	{attribute 'TcIecLibraryType'}
	{attribute 'external_name' := 'F_VN_CreateBandpassButterworthFilter_GUID_D3DC1E0E_00A6_3CD1_3172_0A7CC9A7F473'}
	(* Creates a bandpass Butterworth filter, which can be applied to a frequency domain image by element-wise multiplication. *)
	FUNCTION F_VN_CreateBandpassButterworthFilter : HRESULT
	VAR_INPUT
		ipFilter	:	REFERENCE TO ITcVnImage;	(* Returns the created filter (1 channel of type REAL or LREAL, depending on bDoublePrecision. Non-zero interface pointers are reused.). *)
		nWidth	:	UDINT;	(* Filter width (even, >= 2, must match the width of the image it is applied to) *)
		nHeight	:	UDINT;	(* Filter height (even, >= 2, must match the height of the image it is applied to) *)
		bDoublePrecision	:	BOOL;	(* If true, the filter is generated with double precision (LREAL) instead of single precision (REAL). *)
		bOriginAtCenter	:	BOOL;	(* If true, the filter origin is shifted to the image center. *)
		fCutoffDistance	:	LREAL;	(* The cutoff distance of the Butterworth filter (> 0). *)
		fBandWidth	:	LREAL;	(* The band width of the Butterworth filter (> 0). *)
		nOrder	:	UDINT;	(* The order of the Butterworth filter (> 0). *)
		fScale	:	LREAL;	(* The scale factor of the Butterworth filter denominator term (> 0, e.g. 0.414 or 1.0). *)
		hrPrev	:	HRESULT;	(* HRESULT indicating the result of previous operations (If SUCCEEDED(hrPrev) equals false, no operation is executed.) *)
	END_VAR

END_FUNCTION

// Functions/Fourier Analysis/F_VN_CreateBandpassGaussianFilter

	{attribute 'TcIecLibraryType'}
	{attribute 'external_name' := 'F_VN_CreateBandpassGaussianFilter_GUID_DC938AC3_3255_3FAF_03A0_1C1517F5338C'}
	(* Creates a bandpass Gaussian filter, which can be applied to a frequency domain image by element-wise multiplication. *)
	FUNCTION F_VN_CreateBandpassGaussianFilter : HRESULT
	VAR_INPUT
		ipFilter	:	REFERENCE TO ITcVnImage;	(* Returns the created filter (1 channel of type REAL or LREAL, depending on bDoublePrecision. Non-zero interface pointers are reused.). *)
		nWidth	:	UDINT;	(* Filter width (even, >= 2, must match the width of the image it is applied to) *)
		nHeight	:	UDINT;	(* Filter height (even, >= 2, must match the height of the image it is applied to) *)
		bDoublePrecision	:	BOOL;	(* If true, the filter is generated with double precision (LREAL) instead of single precision (REAL). *)
		bOriginAtCenter	:	BOOL;	(* If true, the filter origin is shifted to the image center. *)
		fCutoffDistance	:	LREAL;	(* The cutoff distance of the Gaussian filter (> 0). *)
		fBandWidth	:	LREAL;	(* The band width of the Gaussian filter (> 0). *)
		hrPrev	:	HRESULT;	(* HRESULT indicating the result of previous operations (If SUCCEEDED(hrPrev) equals false, no operation is executed.) *)
	END_VAR

END_FUNCTION

// Functions/Fourier Analysis/F_VN_CreateBandrejectButterworthFilter

	{attribute 'TcIecLibraryType'}
	{attribute 'external_name' := 'F_VN_CreateBandrejectButterworthFilter_GUID_34508946_AADD_3D36_1DBA_977273E9C532'}
	(* Creates a bandreject Butterworth filter, which can be applied to a frequency domain image by element-wise multiplication. *)
	FUNCTION F_VN_CreateBandrejectButterworthFilter : HRESULT
	VAR_INPUT
		ipFilter	:	REFERENCE TO ITcVnImage;	(* Returns the created filter (1 channel of type REAL or LREAL, depending on bDoublePrecision. Non-zero interface pointers are reused.). *)
		nWidth	:	UDINT;	(* Filter width (even, >= 2, must match the width of the image it is applied to) *)
		nHeight	:	UDINT;	(* Filter height (even, >= 2, must match the height of the image it is applied to) *)
		bDoublePrecision	:	BOOL;	(* If true, the filter is generated with double precision (LREAL) instead of single precision (REAL). *)
		bOriginAtCenter	:	BOOL;	(* If true, the filter origin is shifted to the image center. *)
		fCutoffDistance	:	LREAL;	(* The cutoff distance of the Butterworth filter (> 0). *)
		fBandWidth	:	LREAL;	(* The band width of the Butterworth filter (> 0). *)
		nOrder	:	UDINT;	(* The order of the Butterworth filter (> 0). *)
		fScale	:	LREAL;	(* The scale factor of the Butterworth filter denominator term (> 0, e.g. 0.414 or 1.0). *)
		hrPrev	:	HRESULT;	(* HRESULT indicating the result of previous operations (If SUCCEEDED(hrPrev) equals false, no operation is executed.) *)
	END_VAR

END_FUNCTION

// Functions/Fourier Analysis/F_VN_CreateBandrejectGaussianFilter

	{attribute 'TcIecLibraryType'}
	{attribute 'external_name' := 'F_VN_CreateBandrejectGaussianFilter_GUID_5AAE8B01_5460_3F06_0DD8_D2F7DBC7A3F1'}
	(* Creates a bandreject Gaussian filter, which can be applied to a frequency domain image by element-wise multiplication. *)
	FUNCTION F_VN_CreateBandrejectGaussianFilter : HRESULT
	VAR_INPUT
		ipFilter	:	REFERENCE TO ITcVnImage;	(* Returns the created filter (1 channel of type REAL or LREAL, depending on bDoublePrecision. Non-zero interface pointers are reused.). *)
		nWidth	:	UDINT;	(* Filter width (even, >= 2, must match the width of the image it is applied to) *)
		nHeight	:	UDINT;	(* Filter height (even, >= 2, must match the height of the image it is applied to) *)
		bDoublePrecision	:	BOOL;	(* If true, the filter is generated with double precision (LREAL) instead of single precision (REAL). *)
		bOriginAtCenter	:	BOOL;	(* If true, the filter origin is shifted to the image center. *)
		fCutoffDistance	:	LREAL;	(* The cutoff distance of the Gaussian filter (> 0). *)
		fBandWidth	:	LREAL;	(* The band width of the Gaussian filter (> 0). *)
		hrPrev	:	HRESULT;	(* HRESULT indicating the result of previous operations (If SUCCEEDED(hrPrev) equals false, no operation is executed.) *)
	END_VAR

END_FUNCTION

// Functions/Fourier Analysis/F_VN_CreateHighpassButterworthFilter

	{attribute 'TcIecLibraryType'}
	{attribute 'external_name' := 'F_VN_CreateHighpassButterworthFilter_GUID_519CDF3B_54D9_3152_1A44_7AA98764909A'}
	(* Creates a highpass Butterworth filter, which can be applied to a frequency domain image by element-wise multiplication. *)
	FUNCTION F_VN_CreateHighpassButterworthFilter : HRESULT
	VAR_INPUT
		ipFilter	:	REFERENCE TO ITcVnImage;	(* Returns the created filter (1 channel of type REAL or LREAL, depending on bDoublePrecision. Non-zero interface pointers are reused.). *)
		nWidth	:	UDINT;	(* Filter width (even, >= 2, must match the width of the image it is applied to) *)
		nHeight	:	UDINT;	(* Filter height (even, >= 2, must match the height of the image it is applied to) *)
		bDoublePrecision	:	BOOL;	(* If true, the filter is generated with double precision (LREAL) instead of single precision (REAL). *)
		bOriginAtCenter	:	BOOL;	(* If true, the filter origin is shifted to the image center. *)
		fCutoffDistance	:	LREAL;	(* The cutoff distance of the Butterworth filter (> 0). *)
		nOrder	:	UDINT;	(* The order of the Butterworth filter (> 0). *)
		fScale	:	LREAL;	(* The scale factor of the Butterworth filter denominator term (> 0, e.g. 0.414 or 1.0). *)
		hrPrev	:	HRESULT;	(* HRESULT indicating the result of previous operations (If SUCCEEDED(hrPrev) equals false, no operation is executed.) *)
	END_VAR

END_FUNCTION

// Functions/Fourier Analysis/F_VN_CreateHighpassGaussianFilter

	{attribute 'TcIecLibraryType'}
	{attribute 'external_name' := 'F_VN_CreateHighpassGaussianFilter_GUID_E618411A_DEFA_3D5F_3B14_5E90FD46016B'}
	(* Creates a highpass Gaussian filter, which can be applied to a frequency domain image by element-wise multiplication. *)
	FUNCTION F_VN_CreateHighpassGaussianFilter : HRESULT
	VAR_INPUT
		ipFilter	:	REFERENCE TO ITcVnImage;	(* Returns the created filter (1 channel of type REAL or LREAL, depending on bDoublePrecision. Non-zero interface pointers are reused.). *)
		nWidth	:	UDINT;	(* Filter width (even, >= 2, must match the width of the image it is applied to) *)
		nHeight	:	UDINT;	(* Filter height (even, >= 2, must match the height of the image it is applied to) *)
		bDoublePrecision	:	BOOL;	(* If true, the filter is generated with double precision (LREAL) instead of single precision (REAL). *)
		bOriginAtCenter	:	BOOL;	(* If true, the filter origin is shifted to the image center. *)
		fCutoffDistance	:	LREAL;	(* The cutoff distance of the Gaussian filter (> 0). *)
		hrPrev	:	HRESULT;	(* HRESULT indicating the result of previous operations (If SUCCEEDED(hrPrev) equals false, no operation is executed.) *)
	END_VAR

END_FUNCTION

// Functions/Fourier Analysis/F_VN_CreateLowpassButterworthFilter

	{attribute 'TcIecLibraryType'}
	{attribute 'external_name' := 'F_VN_CreateLowpassButterworthFilter_GUID_409D1272_0EF9_3A29_163E_A5ADC220BBB4'}
	(* Creates a lowpass Butterworth filter, which can be applied to a frequency domain image by element-wise multiplication. *)
	FUNCTION F_VN_CreateLowpassButterworthFilter : HRESULT
	VAR_INPUT
		ipFilter	:	REFERENCE TO ITcVnImage;	(* Returns the created filter (1 channel of type REAL or LREAL, depending on bDoublePrecision. Non-zero interface pointers are reused.). *)
		nWidth	:	UDINT;	(* Filter width (even, >= 2, must match the width of the image it is applied to) *)
		nHeight	:	UDINT;	(* Filter height (even, >= 2, must match the height of the image it is applied to) *)
		bDoublePrecision	:	BOOL;	(* If true, the filter is generated with double precision (LREAL) instead of single precision (REAL). *)
		bOriginAtCenter	:	BOOL;	(* If true, the filter origin is shifted to the image center. *)
		fCutoffDistance	:	LREAL;	(* The cutoff distance of the Butterworth filter (> 0). *)
		nOrder	:	UDINT;	(* The order of the Butterworth filter (> 0). *)
		fScale	:	LREAL;	(* The scale factor of the Butterworth filter denominator term (> 0, e.g. 0.414 or 1.0). *)
		hrPrev	:	HRESULT;	(* HRESULT indicating the result of previous operations (If SUCCEEDED(hrPrev) equals false, no operation is executed.) *)
	END_VAR

END_FUNCTION

// Functions/Fourier Analysis/F_VN_CreateLowpassGaussianFilter

	{attribute 'TcIecLibraryType'}
	{attribute 'external_name' := 'F_VN_CreateLowpassGaussianFilter_GUID_8B9BD84E_306C_3412_3556_4171BB31A9AA'}
	(* Creates a lowpass Gaussian filter, which can be applied to a frequency domain image by element-wise multiplication. *)
	FUNCTION F_VN_CreateLowpassGaussianFilter : HRESULT
	VAR_INPUT
		ipFilter	:	REFERENCE TO ITcVnImage;	(* Returns the created filter (1 channel of type REAL or LREAL, depending on bDoublePrecision. Non-zero interface pointers are reused.). *)
		nWidth	:	UDINT;	(* Filter width (even, >= 2, must match the width of the image it is applied to) *)
		nHeight	:	UDINT;	(* Filter height (even, >= 2, must match the height of the image it is applied to) *)
		bDoublePrecision	:	BOOL;	(* If true, the filter is generated with double precision (LREAL) instead of single precision (REAL). *)
		bOriginAtCenter	:	BOOL;	(* If true, the filter origin is shifted to the image center. *)
		fCutoffDistance	:	LREAL;	(* The cutoff distance of the Gaussian filter (> 0). *)
		hrPrev	:	HRESULT;	(* HRESULT indicating the result of previous operations (If SUCCEEDED(hrPrev) equals false, no operation is executed.) *)
	END_VAR

END_FUNCTION

// Functions/Fourier Analysis/F_VN_Dft

	{attribute 'TcIecLibraryType'}
	{attribute 'external_name' := 'F_VN_Dft_GUID_EB7F674C_B2FA_362B_333C_E819879DB455'}
	(* Computes the DFT for a given image. *)
	FUNCTION F_VN_Dft : HRESULT
	VAR_INPUT
		ipSpatialImage	:	ITcVnImage;	(* Source image (elements of type REAL or LREAL, 1 (Re) or 2 (Re + Im) channels) *)
		ipFrequencyImage	:	REFERENCE TO ITcVnImage;	(* Destination image (same type as ipSpatialImage, but number of channels and size can vary depending on bPackedCCS and bAutoPadding. *)
		bPackedCCS	:	BOOL;	(* If true and ipSpatialImage has only 1 channel, the result image will have 1 channel with packed complex-conjugate-symmetrical format results. Otherwise, the result image will have 2 separate channels (Re + Im), containing the full spectrum. *)
		bAutoPadding	:	BOOL;	(* If true, the input image is automatically padded (with 0s) to optimal size if required, to speed up dft (Creates a temporary copy so that ipSpatialImage content stays unchanged, which also requires some additional computation power. Therefore, it is recommended to compare execution times with and without padding.) *)
		hrPrev	:	HRESULT;	(* HRESULT indicating the result of previous operations (If SUCCEEDED(hrPrev) equals false, no operation is executed.) *)
	END_VAR

END_FUNCTION

// Functions/Fourier Analysis/F_VN_InverseDft

	{attribute 'TcIecLibraryType'}
	{attribute 'external_name' := 'F_VN_InverseDft_GUID_263D4574_0F7D_3790_12C2_708D290903E7'}
	(* Compute the inverse DFT for a given frequency image. *)
	FUNCTION F_VN_InverseDft : HRESULT
	VAR_INPUT
		ipFrequencyImage	:	ITcVnImage;	(* Source frequency image (elements of type REAL or LREAL, 1 (packed CCS) or 2 (Re + Im) channels) *)
		ipSpatialImage	:	REFERENCE TO ITcVnImage;	(* Destination image (Same type as ipFrequencyImage, but number of channels can vary depending on bRealOutput. An appropriate image will be created if required.) *)
		bRealOutput	:	BOOL;	(* Only relevant if ipFrequencyImage has 2 channels. If true, the result image will have only 1 channel. Otherwise, the result image will have 2 separate channels (Re + Im). If ipFrequencyImage has only 1 channel, packed CCS format is assumed and the result image will always have only 1 channel. *)
		hrPrev	:	HRESULT;	(* HRESULT indicating the result of previous operations (If SUCCEEDED(hrPrev) equals false, no operation is executed.) *)
	END_VAR

END_FUNCTION

// Functions/Fourier Analysis/F_VN_OptimalDftSize

	{attribute 'TcIecLibraryType'}
	{attribute 'external_name' := 'F_VN_OptimalDftSize_GUID_08DF2A98_D3C0_3961_2808_BBB884F661F3'}
	(* Computes the optimal image size for applying a dft (can lead to better performance). *)
	FUNCTION F_VN_OptimalDftSize : HRESULT
	VAR_INPUT
		ipImage	:	ITcVnImage;	(* Source image for which to compute the optimal width and height *)
		nOptWidth	:	REFERENCE TO UDINT;	(* Returns the optimal width of the image *)
		nOptHeight	:	REFERENCE TO UDINT;	(* Returns the optimal height of the image *)
		hrPrev	:	HRESULT;	(* HRESULT indicating the result of previous operations (If SUCCEEDED(hrPrev) equals false, no operation is executed.) *)
	END_VAR

END_FUNCTION

// Functions/Fourier Analysis/F_VN_PadImageBorder

	{attribute 'TcIecLibraryType'}
	{attribute 'external_name' := 'F_VN_PadImageBorder_GUID_7562E341_2B8B_34BB_14E9_157BF85E1FEC'}
	(* Add padding (zeros) around the original image borders. *)
	FUNCTION F_VN_PadImageBorder : HRESULT
	VAR_INPUT
		ipSrcImage	:	ITcVnImage;	(* Source image *)
		ipPaddedImage	:	REFERENCE TO ITcVnImage;	(* Padded destination image (Same type as ipSrcImage, an appropriate destination image will be created if required.) *)
		nTopBorder	:	UDINT;	(* Padding height in pixels above top border *)
		nBottomBorder	:	UDINT;	(* Padding height in pixels below bottom border *)
		nLeftBorder	:	UDINT;	(* Padding width in pixels before left border *)
		nRightBorder	:	UDINT;	(* Padding width in pixels after right border *)
		hrPrev	:	HRESULT;	(* HRESULT indicating the result of previous operations (If SUCCEEDED(hrPrev) equals false, no operation is executed.) *)
	END_VAR

END_FUNCTION

// Functions/Fourier Analysis/F_VN_PadImageBorderExp

	{attribute 'TcIecLibraryType'}
	{attribute 'external_name' := 'F_VN_PadImageBorderExp_GUID_D24854F6_1D3E_319C_162B_E66C409C6D41'}
	(* Add padding around the original image borders. (expert function) *)
	FUNCTION F_VN_PadImageBorderExp : HRESULT
	VAR_INPUT
		ipSrcImage	:	ITcVnImage;	(* Source image *)
		ipPaddedImage	:	REFERENCE TO ITcVnImage;	(* Padded destination image (Same type as ipSrcImage, an appropriate destination image will be created if required.) *)
		nTopBorder	:	UDINT;	(* Padding height in pixels above top border *)
		nBottomBorder	:	UDINT;	(* Padding height in pixels below bottom border *)
		nLeftBorder	:	UDINT;	(* Padding width in pixels before left border *)
		nRightBorder	:	UDINT;	(* Padding width in pixels after right border *)
		ePaddingType	:	ETcVnBorderInterpolationMethod;	(* Specifies how the pixel values of the padding area are determined *)
		aPaddingValue	:	REFERENCE TO TcVnVector4_LREAL;	(* Specifies the padding value if CONSTANT is used *)
		hrPrev	:	HRESULT;	(* HRESULT indicating the result of previous operations (If SUCCEEDED(hrPrev) equals false, no operation is executed.) *)
	END_VAR

END_FUNCTION

// Functions/Drawing/F_VN_DrawCircle

	{attribute 'TcIecLibraryType'}
	{attribute 'external_name' := 'F_VN_DrawCircle_GUID_1503D671_B32A_39B0_1A7E_BB6D47FEB820'}
	(* Draws a circle. *)
	FUNCTION F_VN_DrawCircle : HRESULT
	VAR_INPUT
		nCenterX	:	UDINT;	(* x coordinate of the center *)
		nCenterY	:	UDINT;	(* y coordinate of the center *)
		nRadius	:	UDINT;	(* Radius *)
		ipDestImage	:	ITcVnImage;	(* Destination image *)
		aColor	:	REFERENCE TO TcVnVector4_LREAL;	(* Color *)
		nThickness	:	DINT;	(* Line thickness (if negative, the circle is filled) *)
		hrPrev	:	HRESULT;	(* HRESULT indicating the result of previous operations (If SUCCEEDED(hrPrev) equals false, no operation is executed.) *)
	END_VAR

END_FUNCTION

// Functions/Drawing/F_VN_DrawCircleExp

	{attribute 'TcIecLibraryType'}
	{attribute 'external_name' := 'F_VN_DrawCircleExp_GUID_1BBCEDF2_9DF7_3314_302A_7B7B49323D97'}
	(* Draws a circle. *)
	FUNCTION F_VN_DrawCircleExp : HRESULT
	VAR_INPUT
		nCenterX	:	UDINT;	(* x coordinate of the center *)
		nCenterY	:	UDINT;	(* y coordinate of the center *)
		nRadius	:	UDINT;	(* Radius *)
		ipDestImage	:	ITcVnImage;	(* Destination image *)
		aColor	:	REFERENCE TO TcVnVector4_LREAL;	(* Color *)
		nThickness	:	DINT;	(* Line thickness (if negative, the circle is filled) *)
		eLineType	:	ETcVnLineType;	(* Line type *)
		hrPrev	:	HRESULT;	(* HRESULT indicating the result of previous operations (If SUCCEEDED(hrPrev) equals false, no operation is executed.) *)
	END_VAR

END_FUNCTION

// Functions/Drawing/F_VN_DrawCircles

	{attribute 'TcIecLibraryType'}
	{attribute 'external_name' := 'F_VN_DrawCircles_GUID_E3A7DD5D_261F_3C34_1E11_9BA2656FD439'}
	(* Draws circles. *)
	FUNCTION F_VN_DrawCircles : HRESULT
	VAR_INPUT
		ipCircles	:	ITcVnContainer;	(* Container with circles (ContainerType_Vector_TcVnVector3_REAL; Each container element contains the x coordinate of the circle center [0], the y coordinate of the circle center [1], and the radius [2].) *)
		nCircleIndex	:	DINT;	(* Index of a specific circle to be drawn (if negative, all circles within the container are drawn) *)
		ipDestImage	:	ITcVnImage;	(* Destination image *)
		aColor	:	REFERENCE TO TcVnVector4_LREAL;	(* Color *)
		nThickness	:	DINT;	(* Line thickness (if negative, the circle is filled) *)
		hrPrev	:	HRESULT;	(* HRESULT indicating the result of previous operations (If SUCCEEDED(hrPrev) equals false, no operation is executed.) *)
	END_VAR

END_FUNCTION

// Functions/Drawing/F_VN_DrawCirclesExp

	{attribute 'TcIecLibraryType'}
	{attribute 'external_name' := 'F_VN_DrawCirclesExp_GUID_B0C9EA54_3854_3F37_1BB4_4F32EA6C7A2F'}
	(* Draws circles. (expert function) *)
	FUNCTION F_VN_DrawCirclesExp : HRESULT
	VAR_INPUT
		ipCircles	:	ITcVnContainer;	(* Container with circles (ContainerType_Vector_TcVnVector3_REAL; Each container element contains the x coordinate of the circle center [0], the y coordinate of the circle center [1], and the radius [2].) *)
		nCircleIndex	:	DINT;	(* Index of a specific circle to be drawn (if negative, all circles within the container are drawn) *)
		ipDestImage	:	ITcVnImage;	(* Destination image *)
		aColor	:	REFERENCE TO TcVnVector4_LREAL;	(* Color *)
		nThickness	:	DINT;	(* Line thickness (if negative, the circle is filled) *)
		eLineType	:	ETcVnLineType;	(* Line type *)
		hrPrev	:	HRESULT;	(* HRESULT indicating the result of previous operations (If SUCCEEDED(hrPrev) equals false, no operation is executed.) *)
	END_VAR

END_FUNCTION

// Functions/Drawing/F_VN_DrawCircularArc

	{attribute 'TcIecLibraryType'}
	{attribute 'external_name' := 'F_VN_DrawCircularArc_GUID_121719E0_05DB_3D67_0B75_713630B18D92'}
	(* Draws a circular arc. *)
	FUNCTION F_VN_DrawCircularArc : HRESULT
	VAR_INPUT
		stCircularArc	:	REFERENCE TO TcVnCircularArc;	(* Circular arc definition *)
		ipDestImage	:	ITcVnImage;	(* Destination image *)
		aColor	:	REFERENCE TO TcVnVector4_LREAL;	(* Color *)
		nThickness	:	DINT;	(* Line thickness (if negative, the arc is filled) *)
		hrPrev	:	HRESULT;	(* HRESULT indicating the result of previous operations (If SUCCEEDED(hrPrev) equals false, no operation is executed.) *)
	END_VAR

END_FUNCTION

// Functions/Drawing/F_VN_DrawCircularArcExp

	{attribute 'TcIecLibraryType'}
	{attribute 'external_name' := 'F_VN_DrawCircularArcExp_GUID_29FE52B3_2C94_302D_17C7_3DEA0BEF895C'}
	(* Draws a circular arc. (expert function) *)
	FUNCTION F_VN_DrawCircularArcExp : HRESULT
	VAR_INPUT
		stCircularArc	:	REFERENCE TO TcVnCircularArc;	(* Circular arc definition *)
		ipDestImage	:	ITcVnImage;	(* Destination image *)
		aColor	:	REFERENCE TO TcVnVector4_LREAL;	(* Color *)
		nThickness	:	DINT;	(* Line thickness (if negative, the arc is filled) *)
		eLineType	:	ETcVnLineType;	(* Line type *)
		hrPrev	:	HRESULT;	(* HRESULT indicating the result of previous operations (If SUCCEEDED(hrPrev) equals false, no operation is executed.) *)
	END_VAR

END_FUNCTION

// Functions/Drawing/F_VN_DrawContours

	{attribute 'TcIecLibraryType'}
	{attribute 'external_name' := 'F_VN_DrawContours_GUID_4DDB8EE0_9EFD_3D7D_0A1D_A16515665A8A'}
	(* Draws a single point set or multiple point sets that are interpreted as contours. *)
	FUNCTION F_VN_DrawContours : HRESULT
	VAR_INPUT
		ipContours	:	ITcVnContainer;	(* Single contour (ContainerType_Vector_TcVnPoint2_DINT) or multiple contours (ContainerType_Vector_Vector_TcVnPoint2_DINT) *)
		nContourIndex	:	DINT;	(* Index of a specific contour to be drawn (if negative, all contours within the container are drawn) *)
		ipDestImage	:	ITcVnImage;	(* Destination image *)
		aColor	:	REFERENCE TO TcVnVector4_LREAL;	(* Color *)
		nThickness	:	DINT;	(* Line thickness (if negative, the contours are filled) *)
		hrPrev	:	HRESULT;	(* HRESULT indicating the result of previous operations (If SUCCEEDED(hrPrev) equals false, no operation is executed.) *)
	END_VAR

END_FUNCTION

// Functions/Drawing/F_VN_DrawContoursExp

	{attribute 'TcIecLibraryType'}
	{attribute 'external_name' := 'F_VN_DrawContoursExp_GUID_3EB6DE25_2DBC_399F_1688_26782D4E7652'}
	(* Draws a single point set or multiple point sets that are interpreted as contours. (expert function) *)
	FUNCTION F_VN_DrawContoursExp : HRESULT
	VAR_INPUT
		ipContours	:	ITcVnContainer;	(* Single contour (ContainerType_Vector_TcVnPoint2_DINT) or multiple contours (ContainerType_Vector_Vector_TcVnPoint2_DINT) *)
		nContourIndex	:	DINT;	(* Index of a specific contour to be drawn (if negative, all contours within the container are drawn) *)
		ipDestImage	:	ITcVnImage;	(* Destination image *)
		aColor	:	REFERENCE TO TcVnVector4_LREAL;	(* Color *)
		nThickness	:	DINT;	(* Line thickness (if negative, the contours are filled) *)
		eLineType	:	ETcVnLineType;	(* Line type *)
		ipHierarchy	:	ITcVnContainer;	(* Contour hierarchy (ContainerType_Vector_TcVnVector4_DINT) *)
		nMaxLevel	:	DINT;	(* Maximum level of contours to be drawn *)
		aOffset	:	REFERENCE TO TcVnPoint;	(* Offset by which every contour point is shifted *)
		hrPrev	:	HRESULT;	(* HRESULT indicating the result of previous operations (If SUCCEEDED(hrPrev) equals false, no operation is executed.) *)
	END_VAR

END_FUNCTION

// Functions/Drawing/F_VN_DrawEllipse

	{attribute 'TcIecLibraryType'}
	{attribute 'external_name' := 'F_VN_DrawEllipse_GUID_C4C620A7_1B11_32B8_1D39_42E75AB00AD8'}
	(* Draws an ellipse. *)
	FUNCTION F_VN_DrawEllipse : HRESULT
	VAR_INPUT
		stEllipse	:	REFERENCE TO TcVnRotatedRectangle;	(* Ellipse to be drawn (rotation angle in degrees) *)
		ipDestImage	:	ITcVnImage;	(* Destination image *)
		aColor	:	REFERENCE TO TcVnVector4_LREAL;	(* Color *)
		nThickness	:	DINT;	(* Line thickness (if negative, the ellipse is filled) *)
		hrPrev	:	HRESULT;	(* HRESULT indicating the result of previous operations (If SUCCEEDED(hrPrev) equals false, no operation is executed.) *)
	END_VAR

END_FUNCTION

// Functions/Drawing/F_VN_DrawEllipseExp

	{attribute 'TcIecLibraryType'}
	{attribute 'external_name' := 'F_VN_DrawEllipseExp_GUID_35CAB0EB_D927_34D0_3B0E_1CAB03B16108'}
	(* Draws an ellipse. (expert function) *)
	FUNCTION F_VN_DrawEllipseExp : HRESULT
	VAR_INPUT
		stEllipse	:	REFERENCE TO TcVnRotatedRectangle;	(* Ellipse to be drawn (rotation angle in degrees) *)
		ipDestImage	:	ITcVnImage;	(* Destination image *)
		aColor	:	REFERENCE TO TcVnVector4_LREAL;	(* Color *)
		nThickness	:	DINT;	(* Line thickness (if negative, the ellipse is filled) *)
		eLineType	:	ETcVnLineType;	(* Line type *)
		hrPrev	:	HRESULT;	(* HRESULT indicating the result of previous operations (If SUCCEEDED(hrPrev) equals false, no operation is executed.) *)
	END_VAR

END_FUNCTION

// Functions/Drawing/F_VN_DrawKeypoints

	{attribute 'TcIecLibraryType'}
	{attribute 'external_name' := 'F_VN_DrawKeypoints_GUID_8C956DD2_D734_36A5_158B_E1D75DD7AA26'}
	(* Draws the keypoints for visualization purpose. *)
	FUNCTION F_VN_DrawKeypoints : HRESULT
	VAR_INPUT
		ipSrcImage	:	ITcVnImage;	(* Source image (elements of type USINT) *)
		ipKeyPoints	:	ITcVnContainer;	(* Container with the keypoints (ContainerType_Vector_TcVnKeyPoint) *)
		ipDestImage	:	REFERENCE TO ITcVnImage;	(* Destination image (An appropriate image will be created if required.) *)
		hrPrev	:	HRESULT;	(* HRESULT indicating the result of previous operations (If SUCCEEDED(hrPrev) equals false, no operation is executed.) *)
	END_VAR

END_FUNCTION

// Functions/Drawing/F_VN_DrawKeypointsExp

	{attribute 'TcIecLibraryType'}
	{attribute 'external_name' := 'F_VN_DrawKeypointsExp_GUID_22BEE0BC_619E_3666_287B_396FAB7701B1'}
	(* Draws the keypoints for visualization purpose. (expert function) *)
	FUNCTION F_VN_DrawKeypointsExp : HRESULT
	VAR_INPUT
		ipSrcImage	:	ITcVnImage;	(* Source image (elements of type USINT) *)
		ipKeyPoints	:	ITcVnContainer;	(* Container with the keypoints (ContainerType_Vector_TcVnKeyPoint) *)
		ipDestImage	:	REFERENCE TO ITcVnImage;	(* Destination image (An appropriate image will be created if required.) *)
		aColor	:	REFERENCE TO TcVnVector4_LREAL;	(* Color to draw the keypoints (for {-1, -1, -1, -1}, a random color is chosen for each point) *)
		eFlags	:	ETcVnDrawMatchesFlags;	(* A combination of flags to support overdrawing an existing destination image and/or drawing additional (Rich-)Keypoint information (size and orientation) *)
		hrPrev	:	HRESULT;	(* HRESULT indicating the result of previous operations (If SUCCEEDED(hrPrev) equals false, no operation is executed.) *)
	END_VAR

END_FUNCTION

// Functions/Drawing/F_VN_DrawLine

	{attribute 'TcIecLibraryType'}
	{attribute 'external_name' := 'F_VN_DrawLine_GUID_F23D080B_1C6F_3C6F_2EE8_7CCEA69BF02E'}
	(* Draws a line. *)
	FUNCTION F_VN_DrawLine : HRESULT
	VAR_INPUT
		nX1	:	UDINT;	(* x coordinate of the start point *)
		nY1	:	UDINT;	(* y coordinate of the start point *)
		nX2	:	UDINT;	(* x coordinate of the end point *)
		nY2	:	UDINT;	(* y coordinate of the end point *)
		ipDestImage	:	ITcVnImage;	(* Destination image *)
		aColor	:	REFERENCE TO TcVnVector4_LREAL;	(* Color *)
		nThickness	:	DINT;	(* Line thickness *)
		hrPrev	:	HRESULT;	(* HRESULT indicating the result of previous operations (If SUCCEEDED(hrPrev) equals false, no operation is executed.) *)
	END_VAR

END_FUNCTION

// Functions/Drawing/F_VN_DrawLineExp

	{attribute 'TcIecLibraryType'}
	{attribute 'external_name' := 'F_VN_DrawLineExp_GUID_AA6D4FE9_3506_3F4C_037B_6B5F5D077AB5'}
	(* Draws a line. (expert function) *)
	FUNCTION F_VN_DrawLineExp : HRESULT
	VAR_INPUT
		nX1	:	UDINT;	(* x coordinate of the start point *)
		nY1	:	UDINT;	(* y coordinate of the start point *)
		nX2	:	UDINT;	(* x coordinate of the end point *)
		nY2	:	UDINT;	(* y coordinate of the end point *)
		ipDestImage	:	ITcVnImage;	(* Destination image *)
		aColor	:	REFERENCE TO TcVnVector4_LREAL;	(* Color *)
		nThickness	:	DINT;	(* Line thickness *)
		eLineType	:	ETcVnLineType;	(* Line type *)
		nShift	:	UDINT;	(* Fractional bits of the coordinates (bit shift) *)
		hrPrev	:	HRESULT;	(* HRESULT indicating the result of previous operations (If SUCCEEDED(hrPrev) equals false, no operation is executed.) *)
	END_VAR

END_FUNCTION

// Functions/Drawing/F_VN_DrawLine_TcVnVector4_DINT

	{attribute 'TcIecLibraryType'}
	{attribute 'external_name' := 'F_VN_DrawLine_TcVnVector4_DINT_GUID_7C67F5D0_BCDC_3F7B_2FCC_0356A585124E'}
	(* Draws a line. *)
	FUNCTION F_VN_DrawLine_TcVnVector4_DINT : HRESULT
	VAR_INPUT
		aLine	:	REFERENCE TO TcVnVector4_DINT;	(* The start and end point of a line segment [x1, y1, x2, y2] *)
		ipDestImage	:	ITcVnImage;	(* Destination image *)
		aColor	:	REFERENCE TO TcVnVector4_LREAL;	(* Color *)
		nThickness	:	DINT;	(* Line thickness *)
		hrPrev	:	HRESULT;	(* HRESULT indicating the result of previous operations (If SUCCEEDED(hrPrev) equals false, no operation is executed.) *)
	END_VAR

END_FUNCTION

// Functions/Drawing/F_VN_DrawLineExp_TcVnVector4_DINT

	{attribute 'TcIecLibraryType'}
	{attribute 'external_name' := 'F_VN_DrawLineExp_TcVnVector4_DINT_GUID_1C09A8FC_5986_3737_23F5_0F7C79C34548'}
	(* Draws a line. (expert function) *)
	FUNCTION F_VN_DrawLineExp_TcVnVector4_DINT : HRESULT
	VAR_INPUT
		aLine	:	REFERENCE TO TcVnVector4_DINT;	(* The start and end point of a line segment [x1, y1, x2, y2] *)
		ipDestImage	:	ITcVnImage;	(* Destination image *)
		aColor	:	REFERENCE TO TcVnVector4_LREAL;	(* Color *)
		nThickness	:	DINT;	(* Line thickness *)
		eLineType	:	ETcVnLineType;	(* Line type *)
		nShift	:	UDINT;	(* Fractional bits of the coordinates (bit shift) *)
		hrPrev	:	HRESULT;	(* HRESULT indicating the result of previous operations (If SUCCEEDED(hrPrev) equals false, no operation is executed.) *)
	END_VAR

END_FUNCTION

// Functions/Drawing/F_VN_DrawLine_TcVnVector4_LREAL

	{attribute 'TcIecLibraryType'}
	{attribute 'external_name' := 'F_VN_DrawLine_TcVnVector4_LREAL_GUID_87B9BD2C_3B94_36BD_14C4_F71A434A4EAB'}
	(* Draws a line. *)
	FUNCTION F_VN_DrawLine_TcVnVector4_LREAL : HRESULT
	VAR_INPUT
		aLine	:	REFERENCE TO TcVnVector4_LREAL;	(* The first and second element describe the x and y component of the direction vector. The third and fourth element describe the x and y component of the position vector. *)
		ipDestImage	:	ITcVnImage;	(* Destination image *)
		aColor	:	REFERENCE TO TcVnVector4_LREAL;	(* Color *)
		nThickness	:	DINT;	(* Line thickness *)
		hrPrev	:	HRESULT;	(* HRESULT indicating the result of previous operations (If SUCCEEDED(hrPrev) equals false, no operation is executed.) *)
	END_VAR

END_FUNCTION

// Functions/Drawing/F_VN_DrawLineExp_TcVnVector4_LREAL

	{attribute 'TcIecLibraryType'}
	{attribute 'external_name' := 'F_VN_DrawLineExp_TcVnVector4_LREAL_GUID_3ED0AAED_C87B_378B_178D_33F88B7E15A6'}
	(* Draws a line. (expert function) *)
	FUNCTION F_VN_DrawLineExp_TcVnVector4_LREAL : HRESULT
	VAR_INPUT
		aLine	:	REFERENCE TO TcVnVector4_LREAL;	(* The first and second element describe the x and y component of the direction vector. The third and fourth element describe the x and y component of the position vector. *)
		ipDestImage	:	ITcVnImage;	(* Destination image *)
		aColor	:	REFERENCE TO TcVnVector4_LREAL;	(* Color *)
		nThickness	:	DINT;	(* Line thickness *)
		eLineType	:	ETcVnLineType;	(* Line type *)
		nShift	:	UDINT;	(* Fractional bits of the coordinates (bit shift) *)
		hrPrev	:	HRESULT;	(* HRESULT indicating the result of previous operations (If SUCCEEDED(hrPrev) equals false, no operation is executed.) *)
	END_VAR

END_FUNCTION

// Functions/Drawing/F_VN_DrawLines

	{attribute 'TcIecLibraryType'}
	{attribute 'external_name' := 'F_VN_DrawLines_GUID_085A7EF8_E58B_3744_11BD_188CA86A7683'}
	(* Draws lines. *)
	FUNCTION F_VN_DrawLines : HRESULT
	VAR_INPUT
		ipLines	:	ITcVnContainer;	(* Container with line descriptions (ContainerType_Vector_TcVnVector2_REAL: the distance from the origin [0] in pixels and the rotation angle [1] in radians. ContainerType_Vector_TcVnVector4_LREAL: the first and second element describe the x and y component of a vector collinear to the line. The third and fourth element describe the x and y component of a point on the line. ContainerType_Vector_TcVnVector4_DINT: start and end point [x1, y1, x2, y2]) *)
		nLineIndex	:	DINT;	(* Index of a specific line to be drawn (if negative, all lines within the container are drawn) *)
		ipDestImage	:	ITcVnImage;	(* Destination image *)
		aColor	:	REFERENCE TO TcVnVector4_LREAL;	(* Color *)
		nThickness	:	DINT;	(* Line thickness *)
		hrPrev	:	HRESULT;	(* HRESULT indicating the result of previous operations (If SUCCEEDED(hrPrev) equals false, no operation is executed.) *)
	END_VAR

END_FUNCTION

// Functions/Drawing/F_VN_DrawLinesExp

	{attribute 'TcIecLibraryType'}
	{attribute 'external_name' := 'F_VN_DrawLinesExp_GUID_3349DE23_BA35_3613_01CC_9755E183FDB1'}
	(* Draws lines. (expert function) *)
	FUNCTION F_VN_DrawLinesExp : HRESULT
	VAR_INPUT
		ipLines	:	ITcVnContainer;	(* Container with line descriptions (ContainerType_Vector_TcVnVector2_REAL: the distance from the origin [0] in pixels and the rotation angle [1] in radians. ContainerType_Vector_TcVnVector4_LREAL: the first and second element describe the x and y component of a vector collinear to the line. The third and fourth element describe the x and y component of a point on the line. ContainerType_Vector_TcVnVector4_DINT: start and end point [x1, y1, x2, y2]) *)
		nLineIndex	:	DINT;	(* Index of a specific line to be drawn (if negative, all lines within the container are drawn) *)
		ipDestImage	:	ITcVnImage;	(* Destination image *)
		aColor	:	REFERENCE TO TcVnVector4_LREAL;	(* Color *)
		nThickness	:	DINT;	(* Line thickness *)
		eLineType	:	ETcVnLineType;	(* Line type *)
		nShift	:	UDINT;	(* Fractional bits of the coordinates (bit shift) *)
		hrPrev	:	HRESULT;	(* HRESULT indicating the result of previous operations (If SUCCEEDED(hrPrev) equals false, no operation is executed.) *)
	END_VAR

END_FUNCTION

// Functions/Drawing/F_VN_DrawMatches

	{attribute 'TcIecLibraryType'}
	{attribute 'external_name' := 'F_VN_DrawMatches_GUID_E38753BF_5B6F_36D9_3B59_2ADEFD98D379'}
	(* Draws the keypoints and matches for visualization purpose. *)
	FUNCTION F_VN_DrawMatches : HRESULT
	VAR_INPUT
		ipSrcImage1	:	ITcVnImage;	(* Source image 1 (elements of type USINT) *)
		ipKeyPoints1	:	ITcVnContainer;	(* Container with the keypoints 1 (ContainerType_Vector_TcVnKeyPoint) *)
		ipSrcImage2	:	ITcVnImage;	(* Source image 2 (elements of type USINT) *)
		ipKeyPoints2	:	ITcVnContainer;	(* Container with the keypoints 2 (ContainerType_Vector_TcVnKeyPoint) *)
		ipMatches1To2	:	ITcVnContainer;	(* Container with the descriptor matches (ContainerType_Vector_TcVnDMatch) *)
		ipDestImage	:	REFERENCE TO ITcVnImage;	(* Destination image (An appropriate image will be created if required.) *)
		hrPrev	:	HRESULT;	(* HRESULT indicating the result of previous operations (If SUCCEEDED(hrPrev) equals false, no operation is executed.) *)
	END_VAR

END_FUNCTION

// Functions/Drawing/F_VN_DrawMatchesExp

	{attribute 'TcIecLibraryType'}
	{attribute 'external_name' := 'F_VN_DrawMatchesExp_GUID_A93E32D7_DD34_3609_23B2_7F117D8F5FE2'}
	(* Draws the keypoints and matches for visualization purpose. (expert function) *)
	FUNCTION F_VN_DrawMatchesExp : HRESULT
	VAR_INPUT
		ipSrcImage1	:	ITcVnImage;	(* Source image 1 (elements of type USINT) *)
		ipKeyPoints1	:	ITcVnContainer;	(* Container with the keypoints 1 (ContainerType_Vector_TcVnKeyPoint) *)
		ipSrcImage2	:	ITcVnImage;	(* Source image 2 (elements of type USINT) *)
		ipKeyPoints2	:	ITcVnContainer;	(* Container with the keypoints 2 (ContainerType_Vector_TcVnKeyPoint) *)
		ipMatches1To2	:	ITcVnContainer;	(* Container with the descriptor matches (ContainerType_Vector_TcVnDMatch) *)
		ipDestImage	:	REFERENCE TO ITcVnImage;	(* Destination image (An appropriate image will be created if required.) *)
		aMatchColor	:	REFERENCE TO TcVnVector4_LREAL;	(* Color to draw the matches (for {-1, -1, -1, -1}, a random color is chosen for each point and line) *)
		aSingleColor	:	REFERENCE TO TcVnVector4_LREAL;	(* Color to draw the single keypoints (for {-1, -1, -1, -1}, a random color is chosen for each point) *)
		ipMatchesMask	:	ITcVnContainer;	(* Mask to select the matches to be drawn (ContainerType_Vector_SINT; Set to 0 if all matches should be drawn.) *)
		eFlags	:	ETcVnDrawMatchesFlags;	(* A combination of flags to support overdrawing an existing destination image and/or drawing additional (Rich-)Keypoint information (size and orientation) and/or skipping single keypoints *)
		hrPrev	:	HRESULT;	(* HRESULT indicating the result of previous operations (If SUCCEEDED(hrPrev) equals false, no operation is executed.) *)
	END_VAR

END_FUNCTION

// Functions/Drawing/F_VN_DrawPoint

	{attribute 'TcIecLibraryType'}
	{attribute 'external_name' := 'F_VN_DrawPoint_GUID_84B94371_2ABE_309A_018D_1D206868B3BA'}
	(* Draws a point. *)
	FUNCTION F_VN_DrawPoint : HRESULT
	VAR_INPUT
		nX	:	UDINT;	(* x coordinate of the point *)
		nY	:	UDINT;	(* y coordinate of the point *)
		ipDestImage	:	ITcVnImage;	(* Destination image *)
		eShape	:	ETcVnDrawShape;	(* Point shape *)
		aColor	:	REFERENCE TO TcVnVector4_LREAL;	(* Color *)
		hrPrev	:	HRESULT;	(* HRESULT indicating the result of previous operations (If SUCCEEDED(hrPrev) equals false, no operation is executed.) *)
	END_VAR

END_FUNCTION

// Functions/Drawing/F_VN_DrawPointExp

	{attribute 'TcIecLibraryType'}
	{attribute 'external_name' := 'F_VN_DrawPointExp_GUID_6311D72D_4457_3920_3E92_252432BD7E09'}
	(* Draw a point. (expert function) *)
	FUNCTION F_VN_DrawPointExp : HRESULT
	VAR_INPUT
		nX	:	UDINT;	(* x coordinate of the point *)
		nY	:	UDINT;	(* y coordinate of the point *)
		ipDestImage	:	ITcVnImage;	(* Destination image *)
		eShape	:	ETcVnDrawShape;	(* Point shape *)
		aColor	:	REFERENCE TO TcVnVector4_LREAL;	(* Color *)
		nSize	:	UDINT;	(* Size of the shape (half width) *)
		nThickness	:	DINT;	(* Line thickness (if negative, the shape is filled if it is closed) *)
		eLineType	:	ETcVnLineType;	(* Line type *)
		hrPrev	:	HRESULT;	(* HRESULT indicating the result of previous operations (If SUCCEEDED(hrPrev) equals false, no operation is executed.) *)
	END_VAR

END_FUNCTION

// Functions/Drawing/F_VN_DrawPoints

	{attribute 'TcIecLibraryType'}
	{attribute 'external_name' := 'F_VN_DrawPoints_GUID_89680134_4888_39C2_2838_F383F950B2BB'}
	(* Draw a collection of points. *)
	FUNCTION F_VN_DrawPoints : HRESULT
	VAR_INPUT
		ipPoints	:	ITcVnContainer;	(* Container with TcVnPoint2_DINT or TcVnPoint2_REAL elements *)
		ipDestImage	:	ITcVnImage;	(* Destination image *)
		eShape	:	ETcVnDrawShape;	(* Point shape *)
		aColor	:	REFERENCE TO TcVnVector4_LREAL;	(* Color *)
		hrPrev	:	HRESULT;	(* HRESULT indicating the result of previous operations (If SUCCEEDED(hrPrev) equals false, no operation is executed.) *)
	END_VAR

END_FUNCTION

// Functions/Drawing/F_VN_DrawPointsExp

	{attribute 'TcIecLibraryType'}
	{attribute 'external_name' := 'F_VN_DrawPointsExp_GUID_5B12AEE0_4703_3BBC_38CA_126F394AEC72'}
	(* Draw a collection of points. (expert function) *)
	FUNCTION F_VN_DrawPointsExp : HRESULT
	VAR_INPUT
		ipPoints	:	ITcVnContainer;	(* Container with TcVnPoint2_DINT or TcVnPoint2_REAL elements *)
		ipDestImage	:	ITcVnImage;	(* Destination image *)
		eShape	:	ETcVnDrawShape;	(* Point shape *)
		aColor	:	REFERENCE TO TcVnVector4_LREAL;	(* Color *)
		nSize	:	UDINT;	(* Size of the shape (half width) *)
		nThickness	:	DINT;	(* Line thickness (if negative, the shape is filled if it is closed) *)
		eLineType	:	ETcVnLineType;	(* Line type *)
		hrPrev	:	HRESULT;	(* HRESULT indicating the result of previous operations (If SUCCEEDED(hrPrev) equals false, no operation is executed.) *)
	END_VAR

END_FUNCTION

// Functions/Drawing/F_VN_DrawRectangle

	{attribute 'TcIecLibraryType'}
	{attribute 'external_name' := 'F_VN_DrawRectangle_GUID_A5D61916_048E_39C7_244F_79465651E5AD'}
	(* Draw a rectangle. *)
	FUNCTION F_VN_DrawRectangle : HRESULT
	VAR_INPUT
		nTopLeftX	:	UDINT;	(* x coordinate of the top left corner *)
		nTopLeftY	:	UDINT;	(* y coordinate of the top left corner *)
		nBottomRightX	:	UDINT;	(* x coordinate of the bottom right corner *)
		nBottomRightY	:	UDINT;	(* y coordinate of the bottom right corner *)
		ipDestImage	:	ITcVnImage;	(* Destination image *)
		aColor	:	REFERENCE TO TcVnVector4_LREAL;	(* Color *)
		nThickness	:	DINT;	(* Line thickness (if negative, the rectangle is filled) *)
		hrPrev	:	HRESULT;	(* HRESULT indicating the result of previous operations (If SUCCEEDED(hrPrev) equals false, no operation is executed.) *)
	END_VAR

END_FUNCTION

// Functions/Drawing/F_VN_DrawRectangle_TcVnRectangle_UDINT

	{attribute 'TcIecLibraryType'}
	{attribute 'external_name' := 'F_VN_DrawRectangle_TcVnRectangle_UDINT_GUID_24D23C23_70FE_3B75_1A80_930AB1174081'}
	(* Draw a rectangle. *)
	FUNCTION F_VN_DrawRectangle_TcVnRectangle_UDINT : HRESULT
	VAR_INPUT
		stRectangle	:	REFERENCE TO TcVnRectangle_UDINT;	(* Rectangle to be drawn *)
		ipDestImage	:	ITcVnImage;	(* Destination image *)
		aColor	:	REFERENCE TO TcVnVector4_LREAL;	(* Color *)
		nThickness	:	DINT;	(* Line thickness (if negative, the rectangle is filled) *)
		hrPrev	:	HRESULT;	(* HRESULT indicating the result of previous operations (If SUCCEEDED(hrPrev) equals false, no operation is executed.) *)
	END_VAR

END_FUNCTION

// Functions/Drawing/F_VN_DrawRotatedRectangle

	{attribute 'TcIecLibraryType'}
	{attribute 'external_name' := 'F_VN_DrawRotatedRectangle_GUID_86BFDE21_C1C0_3D63_2A5B_F6B3A448320E'}
	(* Draw a rectangle. *)
	FUNCTION F_VN_DrawRotatedRectangle : HRESULT
	VAR_INPUT
		stRectangle	:	REFERENCE TO TcVnRotatedRectangle;	(* Rectangle to be drawn (rotation angle in degrees) *)
		ipDestImage	:	ITcVnImage;	(* Destination image *)
		aColor	:	REFERENCE TO TcVnVector4_LREAL;	(* Color *)
		nThickness	:	DINT;	(* Line thickness (if negative, the rectangle is filled) *)
		hrPrev	:	HRESULT;	(* HRESULT indicating the result of previous operations (If SUCCEEDED(hrPrev) equals false, no operation is executed.) *)
	END_VAR

END_FUNCTION

// Functions/Drawing/F_VN_DrawRotatedRectangleExp

	{attribute 'TcIecLibraryType'}
	{attribute 'external_name' := 'F_VN_DrawRotatedRectangleExp_GUID_91A6F3A4_39D1_309E_21E4_D53ADC9B52DA'}
	(* Draw a rectangle. (expert function) *)
	FUNCTION F_VN_DrawRotatedRectangleExp : HRESULT
	VAR_INPUT
		stRectangle	:	REFERENCE TO TcVnRotatedRectangle;	(* Rectangle to be drawn (rotation angle in degrees) *)
		ipDestImage	:	ITcVnImage;	(* Destination image *)
		aColor	:	REFERENCE TO TcVnVector4_LREAL;	(* Color *)
		nThickness	:	DINT;	(* Line thickness (if negative, the rectangle is filled) *)
		eLineType	:	ETcVnLineType;	(* Line type *)
		hrPrev	:	HRESULT;	(* HRESULT indicating the result of previous operations (If SUCCEEDED(hrPrev) equals false, no operation is executed.) *)
	END_VAR

END_FUNCTION

// Functions/Drawing/F_VN_FillCircle

	{attribute 'TcIecLibraryType'}
	{attribute 'external_name' := 'F_VN_FillCircle_GUID_38571F7A_44E4_39F3_1922_28C4CCE7F968'}
	(* Paint a filled circle. *)
	FUNCTION F_VN_FillCircle : HRESULT
	VAR_INPUT
		nCenterX	:	UDINT;	(* x coordinate of the center *)
		nCenterY	:	UDINT;	(* y coordinate of the center *)
		nRadius	:	UDINT;	(* Radius *)
		ipDestImage	:	ITcVnImage;	(* Destination image *)
		aColor	:	REFERENCE TO TcVnVector4_LREAL;	(* Color *)
		hrPrev	:	HRESULT;	(* HRESULT indicating the result of previous operations (If SUCCEEDED(hrPrev) equals false, no operation is executed.) *)
	END_VAR

END_FUNCTION

// Functions/Drawing/F_VN_FillContours

	{attribute 'TcIecLibraryType'}
	{attribute 'external_name' := 'F_VN_FillContours_GUID_F5B7EC52_A68D_37D6_2BF4_838C321BF25B'}
	(* Paint a single point set or multiple point sets that are interpreted as contours. *)
	FUNCTION F_VN_FillContours : HRESULT
	VAR_INPUT
		ipContours	:	ITcVnContainer;	(* Single contour (ContainerType_Vector_TcVnPoint2_DINT) or multiple contours (ContainerType_Vector_Vector_TcVnPoint2_DINT) *)
		nContourIndex	:	DINT;	(* Index of a specific contour to be drawn (if negative, all contours within the container are drawn) *)
		ipDestImage	:	ITcVnImage;	(* Destination image *)
		aColor	:	REFERENCE TO TcVnVector4_LREAL;	(* Color *)
		hrPrev	:	HRESULT;	(* HRESULT indicating the result of previous operations (If SUCCEEDED(hrPrev) equals false, no operation is executed.) *)
	END_VAR

END_FUNCTION

// Functions/Drawing/F_VN_FillEllipse

	{attribute 'TcIecLibraryType'}
	{attribute 'external_name' := 'F_VN_FillEllipse_GUID_3379A48E_2B9F_3C7C_208D_885D6B95A751'}
	(* Paint a filled ellipse. *)
	FUNCTION F_VN_FillEllipse : HRESULT
	VAR_INPUT
		stEllipse	:	REFERENCE TO TcVnRotatedRectangle;	(* Ellipse to be painted (rotation angle in degrees) *)
		ipDestImage	:	ITcVnImage;	(* Destination image *)
		aColor	:	REFERENCE TO TcVnVector4_LREAL;	(* Color *)
		hrPrev	:	HRESULT;	(* HRESULT indicating the result of previous operations (If SUCCEEDED(hrPrev) equals false, no operation is executed.) *)
	END_VAR

END_FUNCTION

// Functions/Drawing/F_VN_FillRectangle

	{attribute 'TcIecLibraryType'}
	{attribute 'external_name' := 'F_VN_FillRectangle_GUID_D95678A0_FD23_3991_1C3E_9BFF7D779F68'}
	(* Paint a filled rectangle. *)
	FUNCTION F_VN_FillRectangle : HRESULT
	VAR_INPUT
		nTopLeftX	:	UDINT;	(* x coordinate of the top left corner *)
		nTopLeftY	:	UDINT;	(* y coordinate of the top left corner *)
		nBottomRightX	:	UDINT;	(* x coordinate of the bottom right corner *)
		nBottomRightY	:	UDINT;	(* y coordinate of the bottom right corner *)
		ipDestImage	:	ITcVnImage;	(* Destination image *)
		aColor	:	REFERENCE TO TcVnVector4_LREAL;	(* Color *)
		hrPrev	:	HRESULT;	(* HRESULT indicating the result of previous operations (If SUCCEEDED(hrPrev) equals false, no operation is executed.) *)
	END_VAR

END_FUNCTION

// Functions/Drawing/F_VN_FillRotatedRectangle

	{attribute 'TcIecLibraryType'}
	{attribute 'external_name' := 'F_VN_FillRotatedRectangle_GUID_6ABBA740_F56E_3B72_200D_3CAD7816027F'}
	(* Paint a filled rectangle. *)
	FUNCTION F_VN_FillRotatedRectangle : HRESULT
	VAR_INPUT
		stRectangle	:	REFERENCE TO TcVnRotatedRectangle;	(* Rectangle to be painted (rotation angle in degrees) *)
		ipDestImage	:	ITcVnImage;	(* Destination image *)
		aColor	:	REFERENCE TO TcVnVector4_LREAL;	(* Color *)
		hrPrev	:	HRESULT;	(* HRESULT indicating the result of previous operations (If SUCCEEDED(hrPrev) equals false, no operation is executed.) *)
	END_VAR

END_FUNCTION

// Functions/Drawing/F_VN_PutLabel

	{attribute 'TcIecLibraryType'}
	{attribute 'external_name' := 'F_VN_PutLabel_GUID_C38109F1_FDE1_3896_257E_F3DB9BF9637D'}
	(* Write a label (black text on white background) into an image. *)
	FUNCTION F_VN_PutLabel : HRESULT
	VAR_IN_OUT CONSTANT
		sText	:	STRING;	(* Text *)
	END_VAR
	VAR_INPUT
		ipDestImage	:	ITcVnImage;	(* Destination image *)
		nX	:	UDINT;	(* x coordinate (bottom left) *)
		nY	:	UDINT;	(* y coordinate (bottom left) *)
		fFontScale	:	LREAL;	(* Scaling factor *)
		hrPrev	:	HRESULT;	(* HRESULT indicating the result of previous operations (If SUCCEEDED(hrPrev) equals false, no operation is executed.) *)
	END_VAR

END_FUNCTION

// Functions/Drawing/F_VN_PutLabelExp

	{attribute 'TcIecLibraryType'}
	{attribute 'external_name' := 'F_VN_PutLabelExp_GUID_4D756952_3B1A_3916_03F3_A6AC3EFD653E'}
	(* Write a label (text on unified background) into an image. (expert function) *)
	FUNCTION F_VN_PutLabelExp : HRESULT
	VAR_IN_OUT CONSTANT
		sText	:	STRING;	(* Text *)
	END_VAR
	VAR_INPUT
		ipDestImage	:	ITcVnImage;	(* Destination image *)
		nX	:	UDINT;	(* x coordinate (bottom left) *)
		nY	:	UDINT;	(* y coordinate (bottom left) *)
		fFontScale	:	LREAL;	(* Scaling factor *)
		nThickness	:	UDINT;	(* Line thickness *)
		eFontType	:	ETcVnFontType;	(* Font type *)
		aFontColor	:	REFERENCE TO TcVnVector4_LREAL;	(* Font color *)
		aBackgroundColor	:	REFERENCE TO TcVnVector4_LREAL;	(* Background color *)
		eLineType	:	ETcVnLineType;	(* Line type *)
		hrPrev	:	HRESULT;	(* HRESULT indicating the result of previous operations (If SUCCEEDED(hrPrev) equals false, no operation is executed.) *)
	END_VAR

END_FUNCTION

// Functions/Drawing/F_VN_PutText

	{attribute 'TcIecLibraryType'}
	{attribute 'external_name' := 'F_VN_PutText_GUID_E524421B_3247_37C8_24A0_1C1EF39E787D'}
	(* Write text into an image. *)
	FUNCTION F_VN_PutText : HRESULT
	VAR_IN_OUT CONSTANT
		sText	:	STRING;	(* Text *)
	END_VAR
	VAR_INPUT
		ipDestImage	:	ITcVnImage;	(* Destination image *)
		nX	:	UDINT;	(* x coordinate (bottom left) *)
		nY	:	UDINT;	(* y coordinate (bottom left) *)
		eFontType	:	ETcVnFontType;	(* Font type *)
		fFontScale	:	LREAL;	(* Scaling factor *)
		aColor	:	REFERENCE TO TcVnVector4_LREAL;	(* Text color *)
		hrPrev	:	HRESULT;	(* HRESULT indicating the result of previous operations (If SUCCEEDED(hrPrev) equals false, no operation is executed.) *)
	END_VAR

END_FUNCTION

// Functions/Drawing/F_VN_PutTextExp

	{attribute 'TcIecLibraryType'}
	{attribute 'external_name' := 'F_VN_PutTextExp_GUID_B72D289C_50E5_391F_18CA_10CED4B3DE57'}
	(* Write text into an image. (expert function) *)
	FUNCTION F_VN_PutTextExp : HRESULT
	VAR_IN_OUT CONSTANT
		sText	:	STRING;	(* Text *)
	END_VAR
	VAR_INPUT
		ipDestImage	:	ITcVnImage;	(* Destination image *)
		nX	:	UDINT;	(* x coordinate (bottom left) *)
		nY	:	UDINT;	(* y coordinate (bottom left) *)
		eFontType	:	ETcVnFontType;	(* Font type *)
		fFontScale	:	LREAL;	(* Scaling factor *)
		aColor	:	REFERENCE TO TcVnVector4_LREAL;	(* Text color *)
		nThickness	:	DINT;	(* Line thickness *)
		eLineType	:	ETcVnLineType;	(* Line type *)
		bBottomLeftOrigin	:	BOOL;	(* Sets the image origin to the bottom left corner, if true *)
		hrPrev	:	HRESULT;	(* HRESULT indicating the result of previous operations (If SUCCEEDED(hrPrev) equals false, no operation is executed.) *)
	END_VAR

END_FUNCTION

// Functions/Keypoint Features/F_VN_FilterGoodMatches

	{attribute 'TcIecLibraryType'}
	{attribute 'external_name' := 'F_VN_FilterGoodMatches_GUID_70000DF2_87FF_3CD0_0BE1_482B95484E55'}
	(* Filter the descriptor matches and return only good ones. *)
	FUNCTION F_VN_FilterGoodMatches : HRESULT
	VAR_INPUT
		ipMatches	:	ITcVnContainer;	(* Container with descriptor matches (ContainerType_Vector_TcVnDMatch or ContainerType_Vector_Vector_TcVnDMatch) *)
		ipGoodMatches	:	REFERENCE TO ITcVnContainer;	(* Returns a container with good matches (ContainerType_Vector_TcVnDMatch) *)
		fMaxDist	:	REAL;	(* Maximum allowed descriptor distance (-1 disables this filter criterion) *)
		fMaxKnnRatio	:	REAL;	(* Maximum allowed distance ratio between first and second best match ([0..1], used for knn match results only, -1 disables this filter criterion) *)
		hrPrev	:	HRESULT;	(* HRESULT indicating the result of previous operations (If SUCCEEDED(hrPrev) equals false, no operation is executed.) *)
	END_VAR

END_FUNCTION

// Functions/Keypoint Features/F_VN_FindReferenceKeyPointsInImage

	{attribute 'TcIecLibraryType'}
	{attribute 'external_name' := 'F_VN_FindReferenceKeyPointsInImage_GUID_715989BA_AC53_3ABF_127F_9A99CDC0AE7B'}
	(* Searches a reference image, represented by its keypoints and corresponding descriptors, in a given source image. *)
	FUNCTION F_VN_FindReferenceKeyPointsInImage : HRESULT
	VAR_INPUT
		ipSrcKeyPoints	:	ITcVnContainer;	(* KeyPoints of the source image, e.g. (ContainerType_Vector_TcVnKeyPoint) *)
		ipSrcDescriptors	:	ITcVnImage;	(* Descriptors of the source image KeyPoints *)
		ipRefKeyPoints	:	ITcVnContainer;	(* KeyPoints of the reference image, e.g. (ContainerType_Vector_TcVnKeyPoint) *)
		ipRefDescriptors	:	ITcVnImage;	(* Descriptors of the reference image KeyPoints *)
		nRefImageWidth	:	UDINT;	(* Width of the reference image in pixels *)
		nRefImageHeight	:	UDINT;	(* Height of the reference image in pixels *)
		ipEdgePoints	:	REFERENCE TO ITcVnContainer;	(* Returns a container with the 4 edge points of the reference image transformed into the coordinates of the source image (ContainerType_Vector_TcVnPoint2_REAL) *)
		fMaxDist	:	REAL;	(* Maximum allowed descriptor distance (-1 disables this filter criterion) *)
		fMaxKnnRatio	:	REAL;	(* Maximum allowed distance ratio between first and second best match ([0..1], -1 disables this filter criterion) *)
		eNormType	:	ETcVnNormalizationType;	(* Normalization type used for descriptor matching (HAMMING recommended for AKAZE, ORB, and BRISK. HAMMING2 is recommended for ORB if the ORB nBriefPoints parameter is 3 or 4. ) *)
		hrPrev	:	HRESULT;	(* HRESULT indicating the result of previous operations (If SUCCEEDED(hrPrev) equals false, no operation is executed.) *)
	END_VAR
	VAR_OUTPUT
		aPerspectiveTransform	:	TcVnMatrix3x3_LREAL;	(* Returns the perspective transformation matrix, which transforms the reference points to the source points *)
		nNumberOfGoodMatches	:	UDINT;	(* Return the number of good matches *)
		nNumberOfInliers	:	UDINT;	(* Return the number of inlier matches *)
	END_VAR

END_FUNCTION

// Functions/Keypoint Features/F_VN_FindReferenceKeyPointsInImageExp

	{attribute 'TcIecLibraryType'}
	{attribute 'external_name' := 'F_VN_FindReferenceKeyPointsInImageExp_GUID_353A7665_86A6_3A7B_2EEB_DB4B66A97669'}
	(* Searches a reference image, represented by its keypoints and corresponding descriptors, in a given source image. (expert function) *)
	FUNCTION F_VN_FindReferenceKeyPointsInImageExp : HRESULT
	VAR_INPUT
		ipSrcKeyPoints	:	ITcVnContainer;	(* KeyPoints of the source image, e.g. (ContainerType_Vector_TcVnKeyPoint) *)
		ipSrcDescriptors	:	ITcVnImage;	(* Descriptors of the source image KeyPoints *)
		ipRefKeyPoints	:	ITcVnContainer;	(* KeyPoints of the reference image (ContainerType_Vector_TcVnKeyPoint) *)
		ipRefDescriptors	:	ITcVnImage;	(* Descriptors of the reference image KeyPoints *)
		nRefImageWidth	:	UDINT;	(* Width of the reference image in pixels *)
		nRefImageHeight	:	UDINT;	(* Height of the reference image in pixels *)
		ipEdgePoints	:	REFERENCE TO ITcVnContainer;	(* Returns a container with the 4 edge points of the reference image transformed into the coordinates of the source image (ContainerType_Vector_TcVnPoint2_REAL) *)
		fMaxDist	:	REAL;	(* Maximum allowed descriptor distance (-1 disables this filter criterion) *)
		fMaxKnnRatio	:	REAL;	(* Maximum allowed distance ratio between first and second best match ([0..1], -1 disables this filter criterion) *)
		eNormType	:	ETcVnNormalizationType;	(* Normalization type used for descriptor matching (HAMMING recommended for AKAZE, ORB, and BRISK. HAMMING2 is recommended for ORB if the ORB nBriefPoints parameter is 3 or 4. ) *)
		eAlgorithm	:	ETcVnEstimationAlgorithm;	(* Estimation algorithm used for computing the perspective transformation between the two point sets *)
		fReprojThreshold	:	LREAL;	(* Maximum allowed reprojection error to treat a point pair as an inlier (only used if eAlgorithm is RANSAC, RHO) *)
		nMaxIterations	:	UDINT;	(* Maximum number of RANSAC iterations *)
		fConfidence	:	LREAL;	(* Confidence (0..1) *)
		ipGoodMatches	:	REFERENCE TO ITcVnContainer;	(* Returns a container with good matches (optional, set to 0 if not required; ContainerType_Vector_TcVnDMatch) *)
		ipInlierMask	:	REFERENCE TO ITcVnContainer;	(* Returns a mask marking the inliers (optional, set to 0 if not required; ContainerType_Vector_SINT; only for RANSAC, LMEDS) *)
		hrPrev	:	HRESULT;	(* HRESULT indicating the result of previous operations (If SUCCEEDED(hrPrev) equals false, no operation is executed.) *)
	END_VAR
	VAR_OUTPUT
		aPerspectiveTransform	:	TcVnMatrix3x3_LREAL;	(* Returns the perspective transformation matrix, which transforms the reference points to the source points  *)
		nNumberOfGoodMatches	:	UDINT;	(* Return the number of good matches *)
		nNumberOfInliers	:	UDINT;	(* Return the number of inlier matches *)
	END_VAR

END_FUNCTION

// Functions/Keypoint Features/F_VN_FindReferenceKeyPointsInImageAKAZE

	{attribute 'TcIecLibraryType'}
	{attribute 'external_name' := 'F_VN_FindReferenceKeyPointsInImageAKAZE_GUID_49CD3E58_7195_31C7_265F_DB062A50F285'}
	(* Searches a reference image, represented by its AKAZE keypoints and corresponding descriptors, in a given source image (uses the default TcVnParamsAKAZE parameters). *)
	FUNCTION F_VN_FindReferenceKeyPointsInImageAKAZE : HRESULT
	VAR_INPUT
		ipSrcImage	:	ITcVnImage;	(* Source image *)
		ipRefKeyPoints	:	ITcVnContainer;	(* KeyPoints of the reference image, e.g. computed with F_VN_KeyPointsAndDescriptorsAKAZE (ContainerType_Vector_TcVnKeyPoint) *)
		ipRefDescriptors	:	ITcVnImage;	(* Descriptors of the reference image KeyPoints, e.g. computed with F_VN_KeyPointsAndDescriptorsAKAZE *)
		nRefImageWidth	:	UDINT;	(* Width of the reference image in pixels *)
		nRefImageHeight	:	UDINT;	(* Height of the reference image in pixels *)
		ipEdgePoints	:	REFERENCE TO ITcVnContainer;	(* Returns a container with the 4 edge points of the reference image transformed into ipSrcImage coordinates (ContainerType_Vector_TcVnPoint2_REAL) *)
		fMaxDist	:	REAL;	(* Maximum allowed descriptor distance (-1 disables this filter criterion) *)
		fMaxKnnRatio	:	REAL;	(* Maximum allowed distance ratio between first and second best match ([0..1], -1 disables this filter criterion) *)
		hrPrev	:	HRESULT;	(* HRESULT indicating the result of previous operations (If SUCCEEDED(hrPrev) equals false, no operation is executed.) *)
	END_VAR
	VAR_OUTPUT
		aPerspectiveTransform	:	TcVnMatrix3x3_LREAL;	(* Returns the perspective transformation matrix, which transforms the reference points to the source points *)
		nNumberOfGoodMatches	:	UDINT;	(* Return the number of good matches *)
		nNumberOfInliers	:	UDINT;	(* Return the number of inlier matches *)
	END_VAR

END_FUNCTION

// Functions/Keypoint Features/F_VN_KeyPointsAndDescriptorsAKAZE

	{attribute 'TcIecLibraryType'}
	{attribute 'external_name' := 'F_VN_KeyPointsAndDescriptorsAKAZE_GUID_C3B1C953_5A03_3238_18B1_07CC6916DD0D'}
	(* Detects keypoints and compute descriptors using the AKAZE method. *)
	FUNCTION F_VN_KeyPointsAndDescriptorsAKAZE : HRESULT
	VAR_INPUT
		ipSrcImage	:	ITcVnImage;	(* Source image *)
		ipKeyPoints	:	REFERENCE TO ITcVnContainer;	(* Returns a container which is filled with the keypoints (ContainerType_Vector_TcVnKeyPoint; Non-zero interface pointers are reused.) *)
		ipDescriptors	:	REFERENCE TO ITcVnImage;	(* Descriptor image (set to 0 if not required; 1 descriptor in each row; An appropriate image will be created if required.) *)
		hrPrev	:	HRESULT;	(* HRESULT indicating the result of previous operations (If SUCCEEDED(hrPrev) equals false, no operation is executed.) *)
	END_VAR

END_FUNCTION

// Functions/Keypoint Features/F_VN_FindReferenceKeyPointsInImageAKAZEExp

	{attribute 'TcIecLibraryType'}
	{attribute 'external_name' := 'F_VN_FindReferenceKeyPointsInImageAKAZEExp_GUID_AA6D847C_3132_3A9F_3390_4A95C7D8374B'}
	(* Searches a reference image, represented by its AKAZE keypoints and corresponding descriptors, in a given source image. (expert function) *)
	FUNCTION F_VN_FindReferenceKeyPointsInImageAKAZEExp : HRESULT
	VAR_INPUT
		ipSrcImage	:	ITcVnImage;	(* Source image *)
		ipRefKeyPoints	:	ITcVnContainer;	(* KeyPoints of the reference image, e.g. computed with F_VN_KeyPointsAndDescriptorsAKAZE (ContainerType_Vector_TcVnKeyPoint) *)
		ipRefDescriptors	:	ITcVnImage;	(* Descriptors of the reference image KeyPoints, e.g. computed with F_VN_KeyPointsAndDescriptorsAKAZE *)
		nRefImageWidth	:	UDINT;	(* Width of the reference image in pixels *)
		nRefImageHeight	:	UDINT;	(* Height of the reference image in pixels *)
		ipEdgePoints	:	REFERENCE TO ITcVnContainer;	(* Returns a container with the 4 edge points of the reference image transformed into ipSrcImage coordinates (ContainerType_Vector_TcVnPoint2_REAL) *)
		fMaxDist	:	REAL;	(* Maximum allowed descriptor distance (-1 disables this filter criterion) *)
		fMaxKnnRatio	:	REAL;	(* Maximum allowed distance ratio between first and second best match ([0..1], -1 disables this filter criterion) *)
		eNormType	:	ETcVnNormalizationType;	(* Normalization type used for descriptor matching *)
		ipSrcImageMask	:	ITcVnImage;	(* Mask to specify, where to look for keypoints in ipSrcImage (set to 0 if no mask required) *)
		stAkazeParams	:	REFERENCE TO TcVnParamsAKAZE;	(* Parameters to configure the keypoint and descriptor computation for ipSrcImage (resulting descriptors must be compatible to ipRefDescriptors!) *)
		eAlgorithm	:	ETcVnEstimationAlgorithm;	(* Estimation algorithm used for computing the perspective transformation between the two point sets *)
		fReprojThreshold	:	LREAL;	(* Maximum allowed reprojection error to treat a point pair as an inlier (only used if eAlgorithm is RANSAC, RHO) *)
		nMaxIterations	:	UDINT;	(* Maximum number of RANSAC iterations *)
		fConfidence	:	LREAL;	(* Confidence (0..1) *)
		hrPrev	:	HRESULT;	(* HRESULT indicating the result of previous operations (If SUCCEEDED(hrPrev) equals false, no operation is executed.) *)
	END_VAR
	VAR_OUTPUT
		aPerspectiveTransform	:	TcVnMatrix3x3_LREAL;	(* Returns the perspective transformation matrix, which transforms the reference points to the source points  *)
		nNumberOfGoodMatches	:	UDINT;	(* Return the number of good matches *)
		nNumberOfInliers	:	UDINT;	(* Return the number of inlier matches *)
	END_VAR

END_FUNCTION

// Functions/Keypoint Features/F_VN_FindReferenceKeyPointsInImageBRISK

	{attribute 'TcIecLibraryType'}
	{attribute 'external_name' := 'F_VN_FindReferenceKeyPointsInImageBRISK_GUID_36F95353_63D1_3E32_19ED_44C566147741'}
	(* Searches a reference image, represented by its BRISK keypoints and corresponding descriptors, in a given source image (uses the default TcVnParamsBRISK parameters). *)
	FUNCTION F_VN_FindReferenceKeyPointsInImageBRISK : HRESULT
	VAR_INPUT
		ipSrcImage	:	ITcVnImage;	(* Source image *)
		ipRefKeyPoints	:	ITcVnContainer;	(* KeyPoints of the reference image, e.g. computed with F_VN_KeyPointsAndDescriptorsBRISK (ContainerType_Vector_TcVnKeyPoint) *)
		ipRefDescriptors	:	ITcVnImage;	(* Descriptors of the reference image KeyPoints, e.g. computed with F_VN_KeyPointsAndDescriptorsBRISK *)
		nRefImageWidth	:	UDINT;	(* Width of the reference image in pixels *)
		nRefImageHeight	:	UDINT;	(* Height of the reference image in pixels *)
		ipEdgePoints	:	REFERENCE TO ITcVnContainer;	(* Returns a container with the 4 edge points of the reference image transformed into ipSrcImage coordinates (ContainerType_Vector_TcVnPoint2_REAL) *)
		fMaxDist	:	REAL;	(* Maximum allowed descriptor distance (-1 disables this filter criterion) *)
		fMaxKnnRatio	:	REAL;	(* Maximum allowed distance ratio between first and second best match ([0..1], -1 disables this filter criterion) *)
		hrPrev	:	HRESULT;	(* HRESULT indicating the result of previous operations (If SUCCEEDED(hrPrev) equals false, no operation is executed.) *)
	END_VAR
	VAR_OUTPUT
		aPerspectiveTransform	:	TcVnMatrix3x3_LREAL;	(* Returns the perspective transformation matrix, which transforms the reference points to the source points  *)
		nNumberOfGoodMatches	:	UDINT;	(* Return the number of good matches *)
		nNumberOfInliers	:	UDINT;	(* Return the number of inlier matches *)
	END_VAR

END_FUNCTION

// Functions/Keypoint Features/F_VN_KeyPointsAndDescriptorsBRISK

	{attribute 'TcIecLibraryType'}
	{attribute 'external_name' := 'F_VN_KeyPointsAndDescriptorsBRISK_GUID_748D8FDF_FFCD_346A_28A4_84900F400E0D'}
	(* Detects keypoints and compute descriptors using the BRISK method. *)
	FUNCTION F_VN_KeyPointsAndDescriptorsBRISK : HRESULT
	VAR_INPUT
		ipSrcImage	:	ITcVnImage;	(* Source image *)
		ipKeyPoints	:	REFERENCE TO ITcVnContainer;	(* Returns a container which is filled with the keypoints (ContainerType_Vector_TcVnKeyPoint; Non-zero interface pointers are reused.) *)
		ipDescriptors	:	REFERENCE TO ITcVnImage;	(* Descriptor image (set to 0 if not required; 1 descriptor in each row; An appropriate image will be created if required.) *)
		hrPrev	:	HRESULT;	(* HRESULT indicating the result of previous operations (If SUCCEEDED(hrPrev) equals false, no operation is executed.) *)
	END_VAR

END_FUNCTION

// Functions/Keypoint Features/F_VN_FindReferenceKeyPointsInImageBRISKExp

	{attribute 'TcIecLibraryType'}
	{attribute 'external_name' := 'F_VN_FindReferenceKeyPointsInImageBRISKExp_GUID_74F5FE31_2BAF_3AEE_3439_6F8A426B4612'}
	(* Searches a reference image, represented by its BRISK keypoints and corresponding descriptors, in a given source image. (expert function) *)
	FUNCTION F_VN_FindReferenceKeyPointsInImageBRISKExp : HRESULT
	VAR_INPUT
		ipSrcImage	:	ITcVnImage;	(* Source image *)
		ipRefKeyPoints	:	ITcVnContainer;	(* KeyPoints of the reference image, e.g. computed with F_VN_KeyPointsAndDescriptorsBRISK (ContainerType_Vector_TcVnKeyPoint) *)
		ipRefDescriptors	:	ITcVnImage;	(* Descriptors of the reference image KeyPoints, e.g. computed with F_VN_KeyPointsAndDescriptorsBRISK *)
		nRefImageWidth	:	UDINT;	(* Width of the reference image in pixels *)
		nRefImageHeight	:	UDINT;	(* Height of the reference image in pixels *)
		ipEdgePoints	:	REFERENCE TO ITcVnContainer;	(* Returns a container with the 4 edge points of the reference image transformed into ipSrcImage coordinates (ContainerType_Vector_TcVnPoint2_REAL) *)
		fMaxDist	:	REAL;	(* Maximum allowed descriptor distance (-1 disables this filter criterion) *)
		fMaxKnnRatio	:	REAL;	(* Maximum allowed distance ratio between first and second best match ([0..1], -1 disables this filter criterion) *)
		eNormType	:	ETcVnNormalizationType;	(* Normalization type used for descriptor matching *)
		ipSrcImageMask	:	ITcVnImage;	(* Mask to specify, where to look for keypoints in ipSrcImage (set to 0 if no mask required) *)
		stBriskParams	:	REFERENCE TO TcVnParamsBRISK;	(* Parameters to configure the keypoint and descriptor computation for ipSrcImage (resulting descriptors must be compatible to ipRefDescriptors!) *)
		eAlgorithm	:	ETcVnEstimationAlgorithm;	(* Estimation algorithm used for computing the perspective transformation between the two point sets *)
		fReprojThreshold	:	LREAL;	(* Maximum allowed reprojection error to treat a point pair as an inlier (only used if eAlgorithm is RANSAC, RHO) *)
		nMaxIterations	:	UDINT;	(* Maximum number of RANSAC iterations *)
		fConfidence	:	LREAL;	(* Confidence (0..1) *)
		hrPrev	:	HRESULT;	(* HRESULT indicating the result of previous operations (If SUCCEEDED(hrPrev) equals false, no operation is executed.) *)
	END_VAR
	VAR_OUTPUT
		aPerspectiveTransform	:	TcVnMatrix3x3_LREAL;	(* Returns the perspective transformation matrix, which transforms the reference points to the source points  *)
		nNumberOfGoodMatches	:	UDINT;	(* Return the number of good matches *)
		nNumberOfInliers	:	UDINT;	(* Return the number of inlier matches *)
	END_VAR

END_FUNCTION

// Functions/Keypoint Features/F_VN_FindReferenceKeyPointsInImageORB

	{attribute 'TcIecLibraryType'}
	{attribute 'external_name' := 'F_VN_FindReferenceKeyPointsInImageORB_GUID_57B88CC3_5094_308C_1ED8_54ACC8A211FD'}
	(* Searches a reference image, represented by its ORB keypoints and corresponding descriptors, in a given source image (uses the default TcVnParamsORB parameters). *)
	FUNCTION F_VN_FindReferenceKeyPointsInImageORB : HRESULT
	VAR_INPUT
		ipSrcImage	:	ITcVnImage;	(* Source image *)
		ipRefKeyPoints	:	ITcVnContainer;	(* KeyPoints of the reference image, e.g. computed with F_VN_KeyPointsAndDescriptorsORB (ContainerType_Vector_TcVnKeyPoint) *)
		ipRefDescriptors	:	ITcVnImage;	(* Descriptors of the reference image KeyPoints, e.g. computed with F_VN_KeyPointsAndDescriptorsORB *)
		nRefImageWidth	:	UDINT;	(* Width of the reference image in pixels *)
		nRefImageHeight	:	UDINT;	(* Height of the reference image in pixels *)
		ipEdgePoints	:	REFERENCE TO ITcVnContainer;	(* Returns a container with the 4 edge points of the reference image transformed into ipSrcImage coordinates (ContainerType_Vector_TcVnPoint2_REAL) *)
		fMaxDist	:	REAL;	(* Maximum allowed descriptor distance (-1 disables this filter criterion) *)
		fMaxKnnRatio	:	REAL;	(* Maximum allowed distance ratio between first and second best match ([0..1], -1 disables this filter criterion) *)
		hrPrev	:	HRESULT;	(* HRESULT indicating the result of previous operations (If SUCCEEDED(hrPrev) equals false, no operation is executed.) *)
	END_VAR
	VAR_OUTPUT
		aPerspectiveTransform	:	TcVnMatrix3x3_LREAL;	(* Returns the perspective transformation matrix, which transforms the reference points to the source points  *)
		nNumberOfGoodMatches	:	UDINT;	(* Return the number of good matches *)
		nNumberOfInliers	:	UDINT;	(* Return the number of inlier matches *)
	END_VAR

END_FUNCTION

// Functions/Keypoint Features/F_VN_KeyPointsAndDescriptorsORB

	{attribute 'TcIecLibraryType'}
	{attribute 'external_name' := 'F_VN_KeyPointsAndDescriptorsORB_GUID_6F1BDBE2_31F9_350D_28B6_A6C26EA28DD5'}
	(* Detects keypoints and compute descriptors using the ORB method. *)
	FUNCTION F_VN_KeyPointsAndDescriptorsORB : HRESULT
	VAR_INPUT
		ipSrcImage	:	ITcVnImage;	(* Source image *)
		ipKeyPoints	:	REFERENCE TO ITcVnContainer;	(* Returns a container which is filled with the keypoints (ContainerType_Vector_TcVnKeyPoint; Non-zero interface pointers are reused.) *)
		ipDescriptors	:	REFERENCE TO ITcVnImage;	(* Descriptor image (set to 0 if not required; 1 descriptor in each row; An appropriate image will be created if required.) *)
		hrPrev	:	HRESULT;	(* HRESULT indicating the result of previous operations (If SUCCEEDED(hrPrev) equals false, no operation is executed.) *)
	END_VAR

END_FUNCTION

// Functions/Keypoint Features/F_VN_FindReferenceKeyPointsInImageORBExp

	{attribute 'TcIecLibraryType'}
	{attribute 'external_name' := 'F_VN_FindReferenceKeyPointsInImageORBExp_GUID_8ABC29AA_0A88_3AED_1D73_48BD75C6961C'}
	(* Searches a reference image, represented by its ORB keypoints and corresponding descriptors, in a given source image. (expert function) *)
	FUNCTION F_VN_FindReferenceKeyPointsInImageORBExp : HRESULT
	VAR_INPUT
		ipSrcImage	:	ITcVnImage;	(* Source image *)
		ipRefKeyPoints	:	ITcVnContainer;	(* KeyPoints of the reference image, e.g. computed with F_VN_KeyPointsAndDescriptorsORB (ContainerType_Vector_TcVnKeyPoint) *)
		ipRefDescriptors	:	ITcVnImage;	(* Descriptors of the reference image KeyPoints, e.g. computed with F_VN_KeyPointsAndDescriptorsORB *)
		nRefImageWidth	:	UDINT;	(* Width of the reference image in pixels *)
		nRefImageHeight	:	UDINT;	(* Height of the reference image in pixels *)
		ipEdgePoints	:	REFERENCE TO ITcVnContainer;	(* Returns a container with the 4 edge points of the reference image transformed into ipSrcImage coordinates (ContainerType_Vector_TcVnPoint2_REAL) *)
		fMaxDist	:	REAL;	(* Maximum allowed descriptor distance (-1 disables this filter criterion) *)
		fMaxKnnRatio	:	REAL;	(* Maximum allowed distance ratio between first and second best match ([0..1], -1 disables this filter criterion) *)
		eNormType	:	ETcVnNormalizationType;	(* Normalization type used for descriptor matching (HAMMING recommended for ORB, HAMMING2 if the ORB nBriefPoints parameter is 3 or 4) *)
		ipSrcImageMask	:	ITcVnImage;	(* Mask to specify, where to look for keypoints in ipSrcImage (set to 0 if no mask required) *)
		stOrbParams	:	REFERENCE TO TcVnParamsORB;	(* Parameters to configure the keypoint and descriptor computation for ipSrcImage (resulting descriptors must be compatible to ipRefDescriptors!) *)
		eAlgorithm	:	ETcVnEstimationAlgorithm;	(* Estimation algorithm used for computing the perspective transformation between the two point sets *)
		fReprojThreshold	:	LREAL;	(* Maximum allowed reprojection error to treat a point pair as an inlier (only used if eAlgorithm is RANSAC, RHO) *)
		nMaxIterations	:	UDINT;	(* Maximum number of RANSAC iterations *)
		fConfidence	:	LREAL;	(* Confidence (0..1) *)
		hrPrev	:	HRESULT;	(* HRESULT indicating the result of previous operations (If SUCCEEDED(hrPrev) equals false, no operation is executed.) *)
	END_VAR
	VAR_OUTPUT
		aPerspectiveTransform	:	TcVnMatrix3x3_LREAL;	(* Returns the perspective transformation matrix, which transforms the reference points to the source points  *)
		nNumberOfGoodMatches	:	UDINT;	(* Return the number of good matches *)
		nNumberOfInliers	:	UDINT;	(* Return the number of inlier matches *)
	END_VAR

END_FUNCTION

// Functions/Keypoint Features/F_VN_GetMatchCoordinates

	{attribute 'TcIecLibraryType'}
	{attribute 'external_name' := 'F_VN_GetMatchCoordinates_GUID_38C12455_02EE_3DC0_1202_4EA2EDCF86E6'}
	(* Return the coordinates of keypoints that match each other. *)
	FUNCTION F_VN_GetMatchCoordinates : HRESULT
	VAR_INPUT
		ipQueryKeyPoints	:	ITcVnContainer;	(* Container with query Keypoints (CTcVnContainer_Vector_TcVnKeyPoint) *)
		ipTrainKeyPoints	:	ITcVnContainer;	(* Container with train Keypoints (CTcVnContainer_Vector_TcVnKeyPoint) *)
		ipMatches	:	ITcVnContainer;	(* Container with matches between query and train Keypoints (CTcVnContainer_Vector_TcVnDMatch). *)
		ipQueryCoordinates	:	REFERENCE TO ITcVnContainer;	(* Returns a container with the coordinates of keypoints from the query Keypoints that exist in ipMatches (CTcVnContainer_Vector_TcVnPoint2_REAL) *)
		ipTrainCoordinates	:	REFERENCE TO ITcVnContainer;	(* Returns a container with the coordinates of keypoints from the training Keypoints that exist in ipMatches (CTcVnContainer_Vector_TcVnPoint2_REAL) *)
		hrPrev	:	HRESULT;	(* HRESULT indicating the result of previous operations (If SUCCEEDED(hrPrev) equals false, no operation is executed.) *)
	END_VAR

END_FUNCTION

// Functions/Keypoint Features/F_VN_KeyPointsAGAST

	{attribute 'TcIecLibraryType'}
	{attribute 'external_name' := 'F_VN_KeyPointsAGAST_GUID_7B50FBEB_2256_3102_29AA_EDC95E481C3F'}
	(* Detects keypoints using the AGAST method. *)
	FUNCTION F_VN_KeyPointsAGAST : HRESULT
	VAR_INPUT
		ipSrcImage	:	ITcVnImage;	(* Source image *)
		ipKeyPoints	:	REFERENCE TO ITcVnContainer;	(* Returns a container which is filled with the keypoints (ContainerType_Vector_TcVnKeyPoint; Non-zero interface pointers are reused.) *)
		hrPrev	:	HRESULT;	(* HRESULT indicating the result of previous operations (If SUCCEEDED(hrPrev) equals false, no operation is executed.) *)
	END_VAR

END_FUNCTION

// Functions/Keypoint Features/F_VN_KeyPointsAGASTExp

	{attribute 'TcIecLibraryType'}
	{attribute 'external_name' := 'F_VN_KeyPointsAGASTExp_GUID_6C2ABAC6_AD9F_3729_1395_6050AA72B850'}
	(* Detects keypoints using the AGAST method. (expert function) *)
	FUNCTION F_VN_KeyPointsAGASTExp : HRESULT
	VAR_INPUT
		ipSrcImage	:	ITcVnImage;	(* Source image *)
		ipKeyPoints	:	REFERENCE TO ITcVnContainer;	(* Returns a container which is filled with the keypoints (ContainerType_Vector_TcVnKeyPoint; Non-zero interface pointers are reused.) *)
		ipMask	:	ITcVnImage;	(* Mask to specify, where to look for keypoints (set to 0 if no mask required) *)
		stParams	:	REFERENCE TO TcVnParamsAGAST;	(* Additional expert parameters *)
		hrPrev	:	HRESULT;	(* HRESULT indicating the result of previous operations (If SUCCEEDED(hrPrev) equals false, no operation is executed.) *)
	END_VAR

END_FUNCTION

// Functions/Keypoint Features/F_VN_KeyPointsAndDescriptorsAKAZEExp

	{attribute 'TcIecLibraryType'}
	{attribute 'external_name' := 'F_VN_KeyPointsAndDescriptorsAKAZEExp_GUID_9BBB0FAB_2E60_386B_2435_6DE7B4E29201'}
	(* Detects keypoints and compute descriptors using the AKAZE method. (expert function) *)
	FUNCTION F_VN_KeyPointsAndDescriptorsAKAZEExp : HRESULT
	VAR_INPUT
		ipSrcImage	:	ITcVnImage;	(* Source image *)
		ipKeyPoints	:	REFERENCE TO ITcVnContainer;	(* Returns a container which is filled with the keypoints (ContainerType_Vector_TcVnKeyPoint; Non-zero interface pointers are reused.) *)
		ipDescriptors	:	REFERENCE TO ITcVnImage;	(* Descriptor image (set to 0 if not required; 1 descriptor in each row; An appropriate image will be created if required.) *)
		ipMask	:	ITcVnImage;	(* Mask to specify, where to look for keypoints (set to 0 if no mask required) *)
		stParams	:	REFERENCE TO TcVnParamsAKAZE;	(* Additional expert parameters *)
		hrPrev	:	HRESULT;	(* HRESULT indicating the result of previous operations (If SUCCEEDED(hrPrev) equals false, no operation is executed.) *)
	END_VAR

END_FUNCTION

// Functions/Keypoint Features/F_VN_KeyPointsAndDescriptorsBRISKExp

	{attribute 'TcIecLibraryType'}
	{attribute 'external_name' := 'F_VN_KeyPointsAndDescriptorsBRISKExp_GUID_2A20FF1E_9DF0_3397_06CB_6D402520528D'}
	(* Detects keypoints and compute descriptors using the BRISK method. (expert function) *)
	FUNCTION F_VN_KeyPointsAndDescriptorsBRISKExp : HRESULT
	VAR_INPUT
		ipSrcImage	:	ITcVnImage;	(* Source image *)
		ipKeyPoints	:	REFERENCE TO ITcVnContainer;	(* Returns a container which is filled with the keypoints (ContainerType_Vector_TcVnKeyPoint; Non-zero interface pointers are reused.) *)
		ipDescriptors	:	REFERENCE TO ITcVnImage;	(* Descriptor image (set to 0 if not required; 1 descriptor in each row; An appropriate image will be created if required.) *)
		ipMask	:	ITcVnImage;	(* Mask to specify, where to look for keypoints (set to 0 if no mask required) *)
		stParams	:	REFERENCE TO TcVnParamsBRISK;	(* Additional expert parameters *)
		hrPrev	:	HRESULT;	(* HRESULT indicating the result of previous operations (If SUCCEEDED(hrPrev) equals false, no operation is executed.) *)
	END_VAR

END_FUNCTION

// Functions/Keypoint Features/F_VN_KeyPointsAndDescriptorsKAZE

	{attribute 'TcIecLibraryType'}
	{attribute 'external_name' := 'F_VN_KeyPointsAndDescriptorsKAZE_GUID_3B330DFC_F28C_3E92_1BB9_2A4A903AD67D'}
	(* Detects keypoints and compute descriptors using the KAZE method. *)
	FUNCTION F_VN_KeyPointsAndDescriptorsKAZE : HRESULT
	VAR_INPUT
		ipSrcImage	:	ITcVnImage;	(* Source image *)
		ipKeyPoints	:	REFERENCE TO ITcVnContainer;	(* Returns a container which is filled with the keypoints (ContainerType_Vector_TcVnKeyPoint; Non-zero interface pointers are reused.) *)
		ipDescriptors	:	REFERENCE TO ITcVnImage;	(* Descriptor image (set to 0 if not required; 1 descriptor in each row; An appropriate image will be created if required.) *)
		hrPrev	:	HRESULT;	(* HRESULT indicating the result of previous operations (If SUCCEEDED(hrPrev) equals false, no operation is executed.) *)
	END_VAR

END_FUNCTION

// Functions/Keypoint Features/F_VN_KeyPointsAndDescriptorsKAZEExp

	{attribute 'TcIecLibraryType'}
	{attribute 'external_name' := 'F_VN_KeyPointsAndDescriptorsKAZEExp_GUID_5B805AA8_9416_32F1_0817_6AC8D67993BD'}
	(* Detects keypoints and compute descriptors using the KAZE method. (expert function) *)
	FUNCTION F_VN_KeyPointsAndDescriptorsKAZEExp : HRESULT
	VAR_INPUT
		ipSrcImage	:	ITcVnImage;	(* Source image *)
		ipKeyPoints	:	REFERENCE TO ITcVnContainer;	(* Returns a container which is filled with the keypoints (ContainerType_Vector_TcVnKeyPoint; Non-zero interface pointers are reused.) *)
		ipDescriptors	:	REFERENCE TO ITcVnImage;	(* Descriptor image (set to 0 if not required; 1 descriptor in each row; An appropriate image will be created if required.) *)
		ipMask	:	ITcVnImage;	(* Mask to specify, where to look for keypoints (set to 0 if no mask required) *)
		stParams	:	REFERENCE TO TcVnParamsKAZE;	(* Additional expert parameters *)
		hrPrev	:	HRESULT;	(* HRESULT indicating the result of previous operations (If SUCCEEDED(hrPrev) equals false, no operation is executed.) *)
	END_VAR

END_FUNCTION

// Functions/Keypoint Features/F_VN_KeyPointsAndDescriptorsORBExp

	{attribute 'TcIecLibraryType'}
	{attribute 'external_name' := 'F_VN_KeyPointsAndDescriptorsORBExp_GUID_1283225A_4409_3D1F_0993_040BF49736ED'}
	(* Detect keypoints and compute descriptors using the ORB method. (expert function) *)
	FUNCTION F_VN_KeyPointsAndDescriptorsORBExp : HRESULT
	VAR_INPUT
		ipSrcImage	:	ITcVnImage;	(* Source image *)
		ipKeyPoints	:	REFERENCE TO ITcVnContainer;	(* Returns a container which is filled with the keypoints (ContainerType_Vector_TcVnKeyPoint; Non-zero interface pointers are reused.) *)
		ipDescriptors	:	REFERENCE TO ITcVnImage;	(* Descriptor image (set to 0 if not required; 1 descriptor in each row; An appropriate image will be created if required.) *)
		ipMask	:	ITcVnImage;	(* Mask to specify, where to look for keypoints (set to 0 if no mask required) *)
		stParams	:	REFERENCE TO TcVnParamsORB;	(* Additional expert parameters *)
		hrPrev	:	HRESULT;	(* HRESULT indicating the result of previous operations (If SUCCEEDED(hrPrev) equals false, no operation is executed.) *)
	END_VAR

END_FUNCTION

// Functions/Keypoint Features/F_VN_KeyPointsFAST

	{attribute 'TcIecLibraryType'}
	{attribute 'external_name' := 'F_VN_KeyPointsFAST_GUID_A38BB2E9_D9A7_3D85_2113_CE1C54938C21'}
	(* Detects keypoints using the FAST method. *)
	FUNCTION F_VN_KeyPointsFAST : HRESULT
	VAR_INPUT
		ipSrcImage	:	ITcVnImage;	(* Source image (single-channel). *)
		ipKeyPoints	:	REFERENCE TO ITcVnContainer;	(* Returns a container which is filled with the keypoints (ContainerType_Vector_TcVnKeyPoint; Non-zero interface pointers are reused.) *)
		hrPrev	:	HRESULT;	(* HRESULT indicating the result of previous operations (If SUCCEEDED(hrPrev) equals false, no operation is executed.) *)
	END_VAR

END_FUNCTION

// Functions/Keypoint Features/F_VN_KeyPointsFASTExp

	{attribute 'TcIecLibraryType'}
	{attribute 'external_name' := 'F_VN_KeyPointsFASTExp_GUID_79511182_CFED_3A31_3EDF_A2EC03EDADD4'}
	(* Detects keypoints using the FAST method. (expert function) *)
	FUNCTION F_VN_KeyPointsFASTExp : HRESULT
	VAR_INPUT
		ipSrcImage	:	ITcVnImage;	(* Source image *)
		ipKeyPoints	:	REFERENCE TO ITcVnContainer;	(* Returns a container which is filled with the keypoints (ContainerType_Vector_TcVnKeyPoint; Non-zero interface pointers are reused.) *)
		ipMask	:	ITcVnImage;	(* Mask to specify, where to look for keypoints (set to 0 if no mask required) *)
		stParams	:	REFERENCE TO TcVnParamsFAST;	(* Additional expert parameters *)
		hrPrev	:	HRESULT;	(* HRESULT indicating the result of previous operations (If SUCCEEDED(hrPrev) equals false, no operation is executed.) *)
	END_VAR

END_FUNCTION

// Functions/Keypoint Features/F_VN_KeyPointsGFTT

	{attribute 'TcIecLibraryType'}
	{attribute 'external_name' := 'F_VN_KeyPointsGFTT_GUID_BB0E5677_4E2E_38E6_1F83_DA108747DAA5'}
	(* Detects keypoints using the GFTT method, which detects strong corners. *)
	FUNCTION F_VN_KeyPointsGFTT : HRESULT
	VAR_INPUT
		ipSrcImage	:	ITcVnImage;	(* Source image *)
		ipKeyPoints	:	REFERENCE TO ITcVnContainer;	(* Returns a container which is filled with the keypoints (ContainerType_Vector_TcVnKeyPoint; Non-zero interface pointers are reused.) *)
		hrPrev	:	HRESULT;	(* HRESULT indicating the result of previous operations (If SUCCEEDED(hrPrev) equals false, no operation is executed.) *)
	END_VAR

END_FUNCTION

// Functions/Keypoint Features/F_VN_KeyPointsGFTTExp

	{attribute 'TcIecLibraryType'}
	{attribute 'external_name' := 'F_VN_KeyPointsGFTTExp_GUID_377043BF_BDF0_3A0C_072C_A2F9A60C05E4'}
	(* Detects keypoints using the GFTT method, which detects strong corners. (expert function) *)
	FUNCTION F_VN_KeyPointsGFTTExp : HRESULT
	VAR_INPUT
		ipSrcImage	:	ITcVnImage;	(* Source image *)
		ipKeyPoints	:	REFERENCE TO ITcVnContainer;	(* Returns a container which is filled with the keypoints (ContainerType_Vector_TcVnKeyPoint; Non-zero interface pointers are reused.) *)
		ipMask	:	ITcVnImage;	(* Mask to specify, where to look for keypoints (set to 0 if no mask required) *)
		stParams	:	REFERENCE TO TcVnParamsGFTT;	(* Additional expert parameters *)
		hrPrev	:	HRESULT;	(* HRESULT indicating the result of previous operations (If SUCCEEDED(hrPrev) equals false, no operation is executed.) *)
	END_VAR

END_FUNCTION

// Functions/Keypoint Features/F_VN_KeyPointsMSER

	{attribute 'TcIecLibraryType'}
	{attribute 'external_name' := 'F_VN_KeyPointsMSER_GUID_C528B1E6_DE9A_3077_1775_394104648032'}
	(* Detects keypoints using the MSER method. *)
	FUNCTION F_VN_KeyPointsMSER : HRESULT
	VAR_INPUT
		ipSrcImage	:	ITcVnImage;	(* Source image *)
		ipKeyPoints	:	REFERENCE TO ITcVnContainer;	(* Returns a container which is filled with the keypoints (ContainerType_Vector_TcVnKeyPoint; Non-zero interface pointers are reused.) *)
		hrPrev	:	HRESULT;	(* HRESULT indicating the result of previous operations (If SUCCEEDED(hrPrev) equals false, no operation is executed.) *)
	END_VAR

END_FUNCTION

// Functions/Keypoint Features/F_VN_KeyPointsMSERExp

	{attribute 'TcIecLibraryType'}
	{attribute 'external_name' := 'F_VN_KeyPointsMSERExp_GUID_37F7E3B2_6CC3_3F7D_2E10_8980E984D01B'}
	(* Detects keypoints using the MSER method. (expert function) *)
	FUNCTION F_VN_KeyPointsMSERExp : HRESULT
	VAR_INPUT
		ipSrcImage	:	ITcVnImage;	(* Source image *)
		ipKeyPoints	:	REFERENCE TO ITcVnContainer;	(* Returns a container which is filled with the keypoints (ContainerType_Vector_TcVnKeyPoint; Non-zero interface pointers are reused.) *)
		ipMask	:	ITcVnImage;	(* Mask to specify, where to look for keypoints (set to 0 if no mask required) *)
		stParams	:	REFERENCE TO TcVnParamsMSER;	(* Additional expert parameters *)
		hrPrev	:	HRESULT;	(* HRESULT indicating the result of previous operations (If SUCCEEDED(hrPrev) equals false, no operation is executed.) *)
	END_VAR

END_FUNCTION

// Functions/Keypoint Features/F_VN_KeyPointsSB

	{attribute 'TcIecLibraryType'}
	{attribute 'external_name' := 'F_VN_KeyPointsSB_GUID_B6E5066B_76ED_377F_3766_8F28E15FDCD2'}
	(* Detects keypoints using a Simple Blob method:
          - several iterations apply different thresholds to source image
          - connected components (blobs) are detected
          - the center and radius of the blobs are returned as keypoints *)
	FUNCTION F_VN_KeyPointsSB : HRESULT
	VAR_INPUT
		ipSrcImage	:	ITcVnImage;	(* Source image *)
		ipKeyPoints	:	REFERENCE TO ITcVnContainer;	(* Returns a container which is filled with the keypoints (ContainerType_Vector_TcVnKeyPoint; Non-zero interface pointers are reused.) *)
		hrPrev	:	HRESULT;	(* HRESULT indicating the result of previous operations (If SUCCEEDED(hrPrev) equals false, no operation is executed.) *)
	END_VAR

END_FUNCTION

// Functions/Keypoint Features/F_VN_KeyPointsSBExp

	{attribute 'TcIecLibraryType'}
	{attribute 'external_name' := 'F_VN_KeyPointsSBExp_GUID_1DE1B05D_9FC7_3E4E_2067_45B9E555B601'}
	(* 
          Detects keypoints using a Simple Blob method (expert function)
          - several iterations apply different thresholds to source image
          - connected components (blobs) are detected
          - the center and radius of the blobs are returned as keypoints
         *)
	FUNCTION F_VN_KeyPointsSBExp : HRESULT
	VAR_INPUT
		ipSrcImage	:	ITcVnImage;	(* Source image *)
		ipKeyPoints	:	REFERENCE TO ITcVnContainer;	(* Returns a container which is filled with the keypoints (ContainerType_Vector_TcVnKeyPoint; Non-zero interface pointers are reused.) *)
		ipMask	:	ITcVnImage;	(* Mask to specify, where to look for keypoints (currently not supported, set to 0) *)
		stParams	:	REFERENCE TO TcVnParamsSB;	(* Several parameters to filter the detected blobs *)
		hrPrev	:	HRESULT;	(* HRESULT indicating the result of previous operations (If SUCCEEDED(hrPrev) equals false, no operation is executed.) *)
	END_VAR

END_FUNCTION

// Functions/Keypoint Features/F_VN_MatchDescriptorsBF

	{attribute 'TcIecLibraryType'}
	{attribute 'external_name' := 'F_VN_MatchDescriptorsBF_GUID_2F83AE29_E61D_3E8F_3BC2_309EFB47372E'}
	(* Match descriptors using a brute force approach. *)
	FUNCTION F_VN_MatchDescriptorsBF : HRESULT
	VAR_INPUT
		ipQueryDescriptors	:	ITcVnImage;	(* Query descriptors *)
		ipTrainDescriptors	:	ITcVnImage;	(* Training descriptors *)
		ipMatches	:	REFERENCE TO ITcVnContainer;	(* Returns a container which is filled with the descriptor matches (ContainerType_Vector_TcVnDMatch; Non-zero interface pointers are reused.) *)
		hrPrev	:	HRESULT;	(* HRESULT indicating the result of previous operations (If SUCCEEDED(hrPrev) equals false, no operation is executed.) *)
	END_VAR

END_FUNCTION

// Functions/Keypoint Features/F_VN_MatchDescriptorsBFExp

	{attribute 'TcIecLibraryType'}
	{attribute 'external_name' := 'F_VN_MatchDescriptorsBFExp_GUID_DE96F548_6252_3426_0061_08C5CE6CCB32'}
	(* Match descriptors using a brute force approach. (expert function) *)
	FUNCTION F_VN_MatchDescriptorsBFExp : HRESULT
	VAR_INPUT
		ipQueryDescriptors	:	ITcVnImage;	(* Query descriptors *)
		ipTrainDescriptors	:	ITcVnImage;	(* Training descriptors *)
		ipMatches	:	REFERENCE TO ITcVnContainer;	(* Returns a container which is filled with the descriptor matches (ContainerType_Vector_TcVnDMatch; Non-zero interface pointers are reused.) *)
		ipMask	:	ITcVnImage;	(* Mask to specify permissable matches, i.e. query[i] can be matched with train[j] only if mask[i][j] != 0 (set to 0 if no mask required) *)
		eNormType	:	ETcVnNormalizationType;	(* Normalization type (only L1, L2, L2SQR, HAMMING, HAMMING2 supported). HAMMING2 should be used for ORB descriptors if the ORB nBriefPoints parameter is 3 or 4) *)
		bCrossCheck	:	BOOL;	(* If true, only consistent matches are returned, i.e. query->train and train->query detect the same match *)
		hrPrev	:	HRESULT;	(* HRESULT indicating the result of previous operations (If SUCCEEDED(hrPrev) equals false, no operation is executed.) *)
	END_VAR

END_FUNCTION

// Functions/Keypoint Features/F_VN_MatchDescriptorsFlannLsh

	{attribute 'TcIecLibraryType'}
	{attribute 'external_name' := 'F_VN_MatchDescriptorsFlannLsh_GUID_F61DAD6B_E015_36A7_1B6C_44DABC541540'}
	(* Match descriptors using a FLANN based approach with LSH index. *)
	FUNCTION F_VN_MatchDescriptorsFlannLsh : HRESULT
	VAR_INPUT
		ipQueryDescriptors	:	ITcVnImage;	(* Query descriptors *)
		ipTrainDescriptors	:	ITcVnImage;	(* Training descriptors *)
		ipMatches	:	REFERENCE TO ITcVnContainer;	(* Returns a container which is filled with the descriptor matches (ContainerType_Vector_TcVnDMatch; Non-zero interface pointers are reused.) *)
		hrPrev	:	HRESULT;	(* HRESULT indicating the result of previous operations (If SUCCEEDED(hrPrev) equals false, no operation is executed.) *)
	END_VAR

END_FUNCTION

// Functions/Keypoint Features/F_VN_MatchDescriptorsFlannLshExp

	{attribute 'TcIecLibraryType'}
	{attribute 'external_name' := 'F_VN_MatchDescriptorsFlannLshExp_GUID_3AA1A12E_038F_374A_0C8B_2F0908B11BCB'}
	(* Match descriptors using a FLANN based approach with LSH index. (expert function) *)
	FUNCTION F_VN_MatchDescriptorsFlannLshExp : HRESULT
	VAR_INPUT
		ipQueryDescriptors	:	ITcVnImage;	(* Query descriptors *)
		ipTrainDescriptors	:	ITcVnImage;	(* Training descriptors *)
		ipMatches	:	REFERENCE TO ITcVnContainer;	(* Returns a container which is filled with the descriptor matches (ContainerType_Vector_TcVnDMatch; Non-zero interface pointers are reused.) *)
		nTableNumber	:	UDINT;	(* Number of tables *)
		nKeySize	:	UDINT;	(* Key size *)
		nMultiProbeLevel	:	UDINT;	(* Multi-probe level *)
		nChecks	:	UDINT;	(* Maximum number of visited leafs when searching for neighbors *)
		hrPrev	:	HRESULT;	(* HRESULT indicating the result of previous operations (If SUCCEEDED(hrPrev) equals false, no operation is executed.) *)
	END_VAR

END_FUNCTION

// Functions/Keypoint Features/F_VN_MatchDescriptorsKnnBF

	{attribute 'TcIecLibraryType'}
	{attribute 'external_name' := 'F_VN_MatchDescriptorsKnnBF_GUID_9F3D8B49_F62A_3931_3329_1056DC13A2AA'}
	(* Match descriptors (k nearest neighbors) using a brute force approach. *)
	FUNCTION F_VN_MatchDescriptorsKnnBF : HRESULT
	VAR_INPUT
		ipQueryDescriptors	:	ITcVnImage;	(* Query descriptors *)
		ipTrainDescriptors	:	ITcVnImage;	(* Training descriptors *)
		ipMatches	:	REFERENCE TO ITcVnContainer;	(* Returns a container which is filled with the descriptor matches (ContainerType_Vector_Vector_TcVnDMatch; Non-zero interface pointers are reused.) *)
		nK	:	UDINT;	(* Number of required best train matches for each query descriptor (i.e. nk := 2) *)
		hrPrev	:	HRESULT;	(* HRESULT indicating the result of previous operations (If SUCCEEDED(hrPrev) equals false, no operation is executed.) *)
	END_VAR

END_FUNCTION

// Functions/Keypoint Features/F_VN_MatchDescriptorsKnnBFExp

	{attribute 'TcIecLibraryType'}
	{attribute 'external_name' := 'F_VN_MatchDescriptorsKnnBFExp_GUID_D34A8A3D_10DC_3231_0BBA_A94DEBAC93BE'}
	(* Match descriptors (k nearest neighbors) using a brute force approach. (expert function) *)
	FUNCTION F_VN_MatchDescriptorsKnnBFExp : HRESULT
	VAR_INPUT
		ipQueryDescriptors	:	ITcVnImage;	(* Query descriptors *)
		ipTrainDescriptors	:	ITcVnImage;	(* Training descriptors *)
		ipMatches	:	REFERENCE TO ITcVnContainer;	(* Returns a container which is filled with the descriptor matches (ContainerType_Vector_Vector_TcVnDMatch; Non-zero interface pointers are reused.) *)
		nK	:	UDINT;	(* Number of required best train matches for each query descriptor (i.e. nk := 2) *)
		ipMask	:	ITcVnImage;	(* Mask to specify permissable matches, i.e. query[i] can be matched with train[j] only if mask[i][j] != 0 (set to 0 if no mask required) *)
		bCompactResult	:	BOOL;	(* If true, matches vector does not contain entries for fully masked-out query descriptors *)
		eNormType	:	ETcVnNormalizationType;	(* Normalization type (only L1, L2, L2SQR, HAMMING, HAMMING2 supported). HAMMING2 should be used for ORB descriptors if the ORB nBriefPoints parameter is 3 or 4) *)
		bCrossCheck	:	BOOL;	(* If true, only consistent matches are returned, i.e. query->train and train->query detect the same match (only used if nK = 1) *)
		hrPrev	:	HRESULT;	(* HRESULT indicating the result of previous operations (If SUCCEEDED(hrPrev) equals false, no operation is executed.) *)
	END_VAR

END_FUNCTION

// Functions/Keypoint Features/F_VN_MatchDescriptorsKnnFlannLsh

	{attribute 'TcIecLibraryType'}
	{attribute 'external_name' := 'F_VN_MatchDescriptorsKnnFlannLsh_GUID_54318FDB_99D6_3940_3D00_20C5A9F25C25'}
	(* Match descriptors (k nearest neighbors) using a FLANN based approach with LSH index. *)
	FUNCTION F_VN_MatchDescriptorsKnnFlannLsh : HRESULT
	VAR_INPUT
		ipQueryDescriptors	:	ITcVnImage;	(* Query descriptors *)
		ipTrainDescriptors	:	ITcVnImage;	(* Training descriptors *)
		ipMatches	:	REFERENCE TO ITcVnContainer;	(* Returns a container which is filled with the descriptor matches (ContainerType_Vector_Vector_TcVnDMatch; Non-zero interface pointers are reused.) *)
		nK	:	UDINT;	(* Number of required best train matches for each query descriptor (i.e. nk := 2) *)
		hrPrev	:	HRESULT;	(* HRESULT indicating the result of previous operations (If SUCCEEDED(hrPrev) equals false, no operation is executed.) *)
	END_VAR

END_FUNCTION

// Functions/Keypoint Features/F_VN_MatchDescriptorsKnnFlannLshExp

	{attribute 'TcIecLibraryType'}
	{attribute 'external_name' := 'F_VN_MatchDescriptorsKnnFlannLshExp_GUID_5889D7E0_D254_3921_2054_359929CE8A7D'}
	(* Match descriptors (k nearest neighbors) using a FLANN based approach with LSH index. (expert function) *)
	FUNCTION F_VN_MatchDescriptorsKnnFlannLshExp : HRESULT
	VAR_INPUT
		ipQueryDescriptors	:	ITcVnImage;	(* Query descriptors *)
		ipTrainDescriptors	:	ITcVnImage;	(* Training descriptors *)
		ipMatches	:	REFERENCE TO ITcVnContainer;	(* Returns a container which is filled with the descriptor matches (ContainerType_Vector_Vector_TcVnDMatch; Non-zero interface pointers are reused.) *)
		nK	:	UDINT;	(* Number of required best train matches for each query descriptor (i.e. nk := 2) *)
		nTableNumber	:	UDINT;	(* Number of tables *)
		nKeySize	:	UDINT;	(* Key size *)
		nMultiProbeLevel	:	UDINT;	(* Multi-probe level *)
		nChecks	:	UDINT;	(* Maximum number of visited leafs when searching for neighbors *)
		hrPrev	:	HRESULT;	(* HRESULT indicating the result of previous operations (If SUCCEEDED(hrPrev) equals false, no operation is executed.) *)
	END_VAR

END_FUNCTION

// Functions/Keypoint Features/F_VN_RegionsMSER

	{attribute 'TcIecLibraryType'}
	{attribute 'external_name' := 'F_VN_RegionsMSER_GUID_C961D2EA_ADCB_3900_249F_F09CADEF1BAA'}
	(* Detects regions using the MSER method. *)
	FUNCTION F_VN_RegionsMSER : HRESULT
	VAR_INPUT
		ipSrcImage	:	ITcVnImage;	(* Source image *)
		ipRegions	:	REFERENCE TO ITcVnContainer;	(* Returns a container which is filled with the region points (ContainerType_Vector_Vector_TcVnPoint2_DINT; Non-zero interface pointers are reused.) *)
		ipBoundingBoxes	:	REFERENCE TO ITcVnContainer;	(* Returns a container which is filled with the region bounding boxes (ContainerType_Vector_TcVnRectangle_DINT; Non-zero interface pointers are reused.) *)
		hrPrev	:	HRESULT;	(* HRESULT indicating the result of previous operations (If SUCCEEDED(hrPrev) equals false, no operation is executed.) *)
	END_VAR

END_FUNCTION

// Functions/Keypoint Features/F_VN_RegionsMSERExp

	{attribute 'TcIecLibraryType'}
	{attribute 'external_name' := 'F_VN_RegionsMSERExp_GUID_789DB75F_7A54_37DC_05BD_89978FF8DADD'}
	(* Detects regions using the MSER method. (expert function) *)
	FUNCTION F_VN_RegionsMSERExp : HRESULT
	VAR_INPUT
		ipSrcImage	:	ITcVnImage;	(* Source image *)
		ipRegions	:	REFERENCE TO ITcVnContainer;	(* Returns a container which is filled with the region points (ContainerType_Vector_Vector_TcVnPoint2_DINT; Non-zero interface pointers are reused.) *)
		ipBoundingBoxes	:	REFERENCE TO ITcVnContainer;	(* Returns a container which is filled with the region bounding boxes (ContainerType_Vector_TcVnRectangle_DINT; Non-zero interface pointers are reused.) *)
		stParams	:	REFERENCE TO TcVnParamsMSER;	(* Additional expert parameters *)
		hrPrev	:	HRESULT;	(* HRESULT indicating the result of previous operations (If SUCCEEDED(hrPrev) equals false, no operation is executed.) *)
	END_VAR

END_FUNCTION

// Functions/Code Reading/F_VN_ReadBarcode

	{attribute 'TcIecLibraryType'}
	{attribute 'external_name' := 'F_VN_ReadBarcode_GUID_E2F5C339_9134_3972_1B43_BA282A82BD67'}
	(* Detect and interpret a 1d barcode within the provided image.
          Can be canceled by Watchdog. *)
	FUNCTION F_VN_ReadBarcode : HRESULT
	VAR_INPUT
		ipSrcImage	:	ITcVnImage;	(* Source image (USINT elements, 1 channel or 3 channel (3 channel input is expected to be RGB and internally converted to Gray)) *)
		ipDecodedData	:	REFERENCE TO ITcVnContainer;	(* Returns the decoded code (ContainerType_Vector_String_SINT) *)
		eBarcodeType	:	UDINT;	(* Types of barcode to search for (ETcVnBarcodeType) *)
		hrPrev	:	HRESULT;	(* HRESULT indicating the result of previous operations (If SUCCEEDED(hrPrev) equals false, no operation is executed.) *)
	END_VAR

END_FUNCTION

// Functions/Code Reading/F_VN_ReadBarcodeExp

	{attribute 'TcIecLibraryType'}
	{attribute 'external_name' := 'F_VN_ReadBarcodeExp_GUID_E87B5582_80AB_334E_29B6_71EE00F383D4'}
	(* Detect and interpret a 1d barcode within the provided image.
          Can be canceled by Watchdog. *)
	FUNCTION F_VN_ReadBarcodeExp : HRESULT
	VAR_INPUT
		ipSrcImage	:	ITcVnImage;	(* Source image (USINT elements, 1 channel or 3 channel (3 channel input is expected to be RGB and internally converted to Gray)) *)
		ipDecodedData	:	REFERENCE TO ITcVnContainer;	(* Returns the decoded code (ContainerType_Vector_String_SINT) *)
		ipContours	:	REFERENCE TO ITcVnContainer;	(* Returns the code positions as contours (ContainerType_Vector_Vector_TcVnPoint2_DINT) *)
		eBarcodeType	:	UDINT;	(* Types of barcode to search for (ETcVnBarcodeType) *)
		nCodeNumber	:	DINT;	(* Number of 1d barcode that should be detected within the provided image (currently only 1 supported). *)
		eSearchDirection	:	ETcVnBarcodeSearchDirection;	(* Barcode search direction. *)
		hrPrev	:	HRESULT;	(* HRESULT indicating the result of previous operations (If SUCCEEDED(hrPrev) equals false, no operation is executed.) *)
	END_VAR

END_FUNCTION

// Functions/Code Reading/F_VN_ReadDataMatrixCode

